CASE iWorkStep OF
	0:		// Powrót do stanu początkowego (ustawienie zmiennych)
		bResetMethod := bQReady := bQBusy := bQError := FALSE;
		IF NOT bLock AND NOT bRelease THEN
			fbTON(IN:= FALSE);
			stInOuts.bAnvilValve := FALSE;
			iWorkStep := 1;
		END_IF
			
	1: 		// Sprawdzenie czy siłowniki są w dobrej pozycji itp.
			IF stInOuts.bLeftActuatorHome AND stInOuts.bRightActuatorHome  THEN
				bQLocked := FALSE;
				iWorkStep := 5;
			END_IF
	
	5:		// Oczekiwanie na nowy rozkaz
			bResetMethod:= bReleaseMethod:= bAuxOperMethod:= bLockMethod := FALSE;
			bQReady := TRUE;
			actCheckForNewOrder();
		
	10:		// Blokowanie kowadła
		IF bEnCheck AND iCtr_SensorWorkVerification > 2 THEN
			nQErrorId := nStFix_NoWeldLock_ErrorCodes.SensorWorkError;
			iWorkStep := 90;
		ELSIF (fbEnclosureSensorFilter.Q OR NOT bEnCheck) AND stInOuts.bLeftActuatorHome AND stInOuts.bRightActuatorHome THEN
			stInOuts.bAnvilValve := TRUE;
			fbTON(IN:= FALSE);
			iWorkStep := 12;	
		ELSIF NOT fbEnclosureSensorFilter.Q AND bEnCheck THEN
			nQErrorId := nStFix_S17EnclosureWelding_ErrorCodes.PartNotDetectedInFixture;
			iWorkStep := 90;
		ELSIF NOT stInOuts.bLeftActuatorHome OR NOT stInOuts.bRightActuatorHome THEN
			nQErrorId := nStFix_S17EnclosureWelding_ErrorCodes.HomePositionMissing;
			iWorkStep := 90;
		END_IF
		
	12: 	// Oczekiwanie na dociśnięcie obudowy
		fbTON(IN:= TRUE,PT:= T#4S);
		IF NOT stInOuts.bLeftActuatorHome AND NOT stInOuts.bRightActuatorHome AND stInOuts.bAnvilBottom THEN	
			bQBusy := FALSE;
			nQErrorId := 0;
			iWorkStep := 5;
		ELSIF fbTON.ET > T#2S AND (stInOuts.bLeftActuatorHome OR stInOuts.bRightActuatorHome) THEN
			nQErrorId := nStFix_S17EnclosureWelding_ErrorCodes.NoMachineReactionOnStartSig;
			iWorkStep := 90;
		ELSIF fbTON.Q THEN
			nQErrorId := nStFix_S17EnclosureWelding_ErrorCodes.TargetPositionTimeout;
			iWorkStep := 90;
		END_IF
		IF iWorkStep <> 12 THEN fbTON(IN:= FALSE); END_IF
		
	20:		// Dodatkowa operacja	
		bPartWelded:= bLastOperStatus;
		IF bEnCheck THEN
			iCtr_SensorWorkVerification := iCtr_SensorWorkVerification + 1;
		END_IF
		bQBusy := FALSE;
		iWorkStep := 5;
		

	30:	// Kowadło zwolnianie
		stInOuts.bAnvilValve:= FALSE;
		fbTON(IN:= FALSE);
		iWorkStep := 32;
		
	32:	// Oczekiwanie na pozycję domową
		fbTON(IN:= TRUE,PT:= T#5S);
		IF stInOuts.bLeftActuatorHome AND stInOuts.bRightActuatorHome AND NOT stInOuts.bAnvilBottom THEN
			bQBusy := FALSE;
			bQLocked := FALSE;		
			iWorkStep := 5;
		ELSIF fbTON.Q THEN
			nQErrorId := nStFix_S17EnclosureWelding_ErrorCodes.BasePositionTimeout;
			iWorkStep := 90;
		END_IF
		IF iWorkStep <> 32 THEN fbTON(IN:= FALSE); END_IF
		
	90:		// Błąd w pracy kowadła
		bQBusy := FALSE;
		bQError := TRUE;
		iWorkStep := 91;
		
	91:
		IF bRelease OR bResetMethod THEN
			iCtr_SensorWorkVerification := 0;
			stInOuts.bAnvilValve := FALSE;
			bQError := FALSE;
			nQErrorId := 0;
			iWorkStep := 0;
		END_IF
		
	ELSE
		mNewEvent(nStFix_S17EnclosureWelding_ErrorCodes.ProgramConfigError);		
END_CASE

END_FUNCTION_BLOCK

// ProdLineMachines/Sonictech/SerialCom/fbSonictechSerialCom
FUNCTION_BLOCK fbSonictechSerialCom IMPLEMENTS I_SonicTech_SerialCom
VAR CONSTANT
	uiMAX_QUEUE_SIZE: UINT := 10;
END_VAR
VAR_IN_OUT
	stData:stSerialComData;
END_VAR
VAR_INPUT
	tTimeout:TIME := T#2S;		// Timeout komunikacji 
	uiResendQty :UINT := 1;			// Liczba ponownych wysłań komend
END_VAR
VAR_OUTPUT
END_VAR
VAR
	fbSerialRead: fbSonictechSerialRcv;
	astCmdsQueue: ARRAY[1..uiMAX_QUEUE_SIZE] OF POINTER TO stSonicTech_SerialCMD;
	bQueueEmpty: BOOL := TRUE;
	bQueueFull: BOOL;
	uiLastCmdIndex: UINT;
	pPtr2ActCmd : POINTER TO stSonicTech_SerialCMD;
	pstDriverData: POINTER TO stSonicTech_SerialStructSoftVer;
	psActProgName: POINTER TO STRING(16);
	pstParametersRange: POINTER TO stSonicTech_SerialStructGenParamsRange;
	pstActualProgramParameters: POINTER TO stSonicTech_SerialStructProgParams;
	pstLastWeldParameters: POINTER TO stSonicTech_SerialStructWeldParams;
	stTestCmdData: stSonicTech_SerialCMD;
	sTestSerialNb: STRING(15);
	stTestDriverData: stSonicTech_SerialStructSoftVer;
	stTestParametersRange: stSonicTech_SerialStructGenParamsRange;
	stTestActualProgramParameters: stSonicTech_SerialStructProgParams;
	stTestLastWeldParameters: stSonicTech_SerialStructWeldParams;
	sTestActProgName: STRING(16);
	byTestActualSonicTechProgNb: BYTE;
	byErrorCode, byTestErrorCode: BYTE;
	// Odbiór danych RS232 
	i: INT;		// Indeks używany w pętlach
	abBufor_Send: ARRAY [1..80] OF BYTE;
	abBufor_String: ARRAY [0..MAX_STRING_LENGTH] OF BYTE;
	bSumaKontrolnaZapytania: BYTE;
	fbSendData:SendData;
	sActProgName2: STRING(16);
	ptPointerToINT:POINTER TO INT;
	ptPointerToUINT:POINTER TO UINT;
	fbTON_RcvTimeout: TON;
	
// Inne	
	nCmdType: nSonicTech_SerialCmdClasses;
	iRozmiarBufora: INT;
	nRecvFrameType: nSonicTech_SerialCmdType;
	bSendCmd: BOOL;				// Bit ustawiany gdy trzeba wysłać rozkaz - kasowany po zakończeniu wysyłania OK bądź NOK
	bWaitingForResponse: BOOL;		// Bit ustawiany po pozytywnym wysłaniu komendy - kasowany po odbiorze danych 
	bReSendCommand: BOOL;		// W razie błędu spróbuj ponownie wysłać komendę
	bCmdExecError: BOOL;	// Błąd w przetwarzaniu komedny
	enComSendErrorMem: Tc2_SerialCom.ComError_t;
	fbClearBuffers:ClearComBuffer;
	bLongExecuteCmd: BOOL;
	fbTONResetComm: TON;
	rCommandReadMeanTime: REAL;
	iComErrors: INT;
	uiReSended: UINT;
	bComReset: BOOL;
	
	bCmdEndedOK: BOOL;
	bAddTestCmd: BOOL;
	nTestCmdType: nSonicTech_SerialCmdClasses;
	fbTON_ComTime: TON;
	bSendTestData: BOOL;
	bPtrsChanged: BOOL;
	bTestCmdFailed: BOOL;
	rLastCmdExecTime: REAL;
	bSendError: BOOL;
	sLastProgName: STRING(255);
	udi_SencCmdCtr: UDINT;
	ui: UINT;
END_VAR

(* ********* Obsługa komunikacji *********
	Nowe zapytanie możliwe gdy typ zapytania=0, jeśli chcemy wykonać zapytanie zmieniamy wartość iTypZapytanie na pożądaną wartość.
	Pętla poniżej zgodnie z typem zapytania przygotowuje zapytanie oraz ustawia flagę bSend.
	Blok wysyłania danych w reakcji na bSend wysyła dane, jeśli wysłanie danych powiodło się, resetuje flagę bSend oraz ustawia bOczekiwanieNaOdpowiedź
	Blok odbierający dane monitoruje zbocze narastające na zmiennej bOczekiwanieNaOdpowiedź, gdy będzie R_TRIG resetuje wewnętrzne dane, ustawia flagę bBusy oraz odbiera dane od zgrzewarki
	Jeśli odbiór był OK wystawia sygnał bDataRecived, jeśli nie wystawia sygnał błędu oraz zeruję flagę bBusy.
*)

ACT_Test_Cmds();
IF nCmdType = nSonicTech_SerialCmdClasses.NoCMD THEN		// Oczekiwanie na nową komendę:
	IF astCmdsQueue[1] <> 0 AND NOT bComReset THEN		// Pobranie nowej komendy z kolejki 
		bLongExecuteCmd := bSendCmd := bWaitingForResponse := FALSE;
		bCmdEndedOK := bCmdExecError := FALSE;
		nCmdType := astCmdsQueue[1]^.nCmdType;
		pPtr2ActCmd := astCmdsQueue[1]; 
		pPtr2ActCmd^.bDone := pPtr2ActCmd^.bError := pPtr2ActCmd^.bSended := FALSE;
	END_IF		
ELSIF bCmdEndedOK OR bCmdExecError THEN			// Sprawdzenie wyniku przetwarzania komendy
	bWaitingForResponse := FALSE;
	fMeanFilter(rInputValue := TIME_TO_REAL(fbTONResetComm.ET), rDelta := 10.0, rMeanValue := rCommandReadMeanTime);
	IF pPtr2ActCmd <> 0 THEN
		pPtr2ActCmd^.bDone := TRUE;
		IF bCmdEndedOK THEN
			pPtr2ActCmd^.nCmdStatus := nSonicTech_SerialCmdStatus.CmdSucceed;
		ELSE
			pPtr2ActCmd^.bError := TRUE;
			pPtr2ActCmd^.nCmdStatus := nSonicTech_SerialCmdStatus.CmdError;	
		END_IF
	END_IF
	pPtr2ActCmd := 0;
	nCmdType := nSonicTech_SerialCmdClasses.NoCMD;
	
	// Sprawdzenie czy są nowe komendy do wykonania
	IF astCmdsQueue[2] <> 0 THEN	// Jest komenda
		MEMMOVE(srcAddr := ADR(astCmdsQueue[2]), destAddr := ADR(astCmdsQueue[1]), n := (uiMAX_QUEUE_SIZE-1)*SIZEOF(astCmdsQueue[2]));
		astCmdsQueue[uiLastCmdIndex]:= 0;
		uiLastCmdIndex := uiLastCmdIndex -1;
		bQueueFull := FALSE;
	ELSE
		astCmdsQueue[1] := 0;
		uiLastCmdIndex := 0;
		bQueueEmpty := TRUE;
	END_IF
END_IF

// Timeout
FOR ui := 2 TO uiLastCmdIndex BY 1 DO
	IF astCmdsQueue[ui] <> 0 THEN
		IF (GVL_Aircom.stAC_DT_Data.tActualTime - astCmdsQueue[ui]^.tTimeStamp) > tTimeout THEN	// Timeout in queue
			astCmdsQueue[ui]^.bDone := astCmdsQueue[ui]^.bError := TRUE;
			astCmdsQueue[ui]^.nCmdStatus := nSonicTech_SerialCmdStatus.CmdError;
			MEMMOVE(srcAddr:= ADR(astCmdsQueue[ui+1]), destAddr := ADR(astCmdsQueue[ui]), n :=(uiLastCmdIndex - ui)*SIZEOF(astCmdsQueue[1]));
			ui := ui -1;	// Ręczna korekta inkrementacji zmiennej w FOR
		END_IF
	END_IF
END_FOR

CASE nCmdType OF
	nSonicTech_SerialCmdClasses.NoCMD:	// Bezczynność
	
	nSonicTech_SerialCmdClasses.ReadSerialNb:	
		IF NOT bSendCmd AND NOT bWaitingForResponse OR bReSendCommand THEN
			abBufor_Send[4]:= 16#00;		// Kod funkcji 0x00 - odczyt numeru seryjnego sterownika
			mFillSendBuffor(Frame := nSonicTech_SerialCmdType.SD1);
			nRecvFrameType := nSonicTech_SerialCmdType.SD2;	
			bSendCmd := TRUE;
		ELSIF fbSerialRead.bDataReceived THEN				// Odbiór danych
			sTestSerialNb := '';
//			fbSerialRead.abBufor_Recv[2] := LIMIT(4,fbSerialRead.abBufor_Recv[2],249);
			IF pPtr2ActCmd <> 0 AND_THEN pPtr2ActCmd^.uiExchangeDataSize >= (fbSerialRead.abBufor_Recv[2]-3) THEN
				MEMCPY(srcAddr := ADR(fbSerialRead.abBufor_Recv[8]),destAddr := pPtr2ActCmd^.pExchangeData, n := (fbSerialRead.abBufor_Recv[2]-3));
				bCmdEndedOK:= TRUE;
			END_IF
			bWaitingForResponse := FALSE;
		END_IF

 	nSonicTech_SerialCmdClasses.ReadMaxParamsValues:	
		IF NOT bSendCmd AND NOT bWaitingForResponse OR bReSendCommand THEN
			abBufor_Send[4]:= 16#01;		// Kod funkcji 0x01 - odczyt zakresu parametrów
			mFillSendBuffor(Frame := nSonicTech_SerialCmdType.SD1);
			nRecvFrameType := nSonicTech_SerialCmdType.SD2;	
			bSendCmd := TRUE;
		ELSIF fbSerialRead.bDataReceived  THEN				// Odbiór danych
			IF pPtr2ActCmd <> 0 AND_THEN pPtr2ActCmd^.uiExchangeDataSize = SIZEOF(stTestParametersRange) THEN
				pstParametersRange := pPtr2ActCmd^.pExchangeData;
				pstParametersRange^.byGeneratorType := fbSerialRead.abBufor_Recv[8];
				ptPointerToUINT := ADR(fbSerialRead.abBufor_Recv[9]);
				pstParametersRange^.uiMinGenFrequency := ROL(ptPointerToUINT^, 8);
				ptPointerToUINT := ADR(fbSerialRead.abBufor_Recv[11]);
				pstParametersRange^.uiMaxGenFrequency := ROL(ptPointerToUINT^, 8);
				ptPointerToUINT := ADR(fbSerialRead.abBufor_Recv[13]);
				pstParametersRange^.uiMaxGenPower := ROL(ptPointerToUINT^, 8);
				ptPointerToUINT := ADR(fbSerialRead.abBufor_Recv[15]);
				pstParametersRange^.uiEncoderLength := ROL(ptPointerToUINT^, 8);
				bCmdEndedOK:= TRUE;
			END_IF
			bWaitingForResponse := FALSE;
		END_IF

	nSonicTech_SerialCmdClasses.ReadSoftVer:	
		IF NOT bSendCmd AND NOT bWaitingForResponse OR bReSendCommand THEN
			abBufor_Send[4]:= 16#03;		// Kod funkcji 0x03 - odczyt wersji oprogramowania
			mFillSendBuffor(Frame := nSonicTech_SerialCmdType.SD1);
			nRecvFrameType := nSonicTech_SerialCmdType.SD3;
			bSendCmd := TRUE;
		ELSIF fbSerialRead.bDataReceived  THEN				// Odbiór danych
			IF pPtr2ActCmd <> 0 AND_THEN pPtr2ActCmd^.uiExchangeDataSize = SIZEOF(stTestDriverData) THEN
				pstDriverData := pPtr2ActCmd^.pExchangeData;
				pstDriverData^.byDriverModel := fbSerialRead.abBufor_Recv[5];
				pstDriverData^.byMajorVersion := fbSerialRead.abBufor_Recv[6];
				pstDriverData^.byMinorVersion := fbSerialRead.abBufor_Recv[7];
				ptPointerToINT := ADR(fbSerialRead.abBufor_Recv[8]);
				pstDriverData^.iBuildNumber := ptPointerToINT^;
				bCmdEndedOK:= TRUE;
			END_IF
		//	sSoftwareVersion := CONCAT(BYTE_TO_STRING(stDaneSterZgrzew.byMajorVersion),CONCAT('.',CONCAT(BYTE_TO_STRING(stDaneSterZgrzew.byMinorVersion),CONCAT('.',INT_TO_STRING(stDaneSterZgrzew.iBuildNumber)))));
			bWaitingForResponse := FALSE;
		END_IF

	nSonicTech_SerialCmdClasses.ReadProgNb:	
		IF NOT bSendCmd AND NOT bWaitingForResponse OR bReSendCommand THEN
			abBufor_Send[4]:= 16#10;		// Kod funkcji 0x10 - odczyt numeru aktualnego programu
			mFillSendBuffor(Frame := nSonicTech_SerialCmdType.SD1);
			nRecvFrameType := nSonicTech_SerialCmdType.SD3;	
			bSendCmd := TRUE;
		ELSIF fbSerialRead.bDataReceived  THEN				// Odbiór danych
			IF pPtr2ActCmd <> 0 AND_THEN pPtr2ActCmd^.uiExchangeDataSize = SIZEOF(byTestActualSonicTechProgNb) THEN
				pPtr2ActCmd^.pExchangeData^ := fbSerialRead.abBufor_Recv[5];
				bCmdEndedOK:= TRUE;
			END_IF
			bWaitingForResponse := FALSE;
		END_IF
			
	nSonicTech_SerialCmdClasses.SetProgNb:
		IF pPtr2ActCmd <> 0 AND_THEN NOT bSendCmd AND NOT bWaitingForResponse OR bReSendCommand THEN
			abBufor_Send[4]:= 16#10;		// Kod funkcji 0x10 - odczyt numeru aktualnego programu
//			MEMCPY(srcAddr := pPtr2ActCmd^.pExchangeData, destAddr := ADR(abBufor_Send[5]) , n := pPtr2ActCmd^.uiExchangeDataSize);
			abBufor_Send[5]:= pPtr2ActCmd^.pExchangeData^;		// Numer aktualnego programu
			MEMSET(destAddr := ADR(abBufor_Send[6]),fillByte:= 0, n:= 7);	// Zerowanie pozostałych bajtów
			mFillSendBuffor(Frame := nSonicTech_SerialCmdType.SD3);
			nRecvFrameType := nSonicTech_SerialCmdType.SC;		
			bSendCmd := TRUE;
		ELSIF fbSerialRead.bDataReceived  THEN				// Odbiór danych
			bCmdEndedOK:= TRUE;
			bWaitingForResponse := FALSE;
		END_IF
			
	nSonicTech_SerialCmdClasses.ReadProgName:
		IF NOT fbSendData.Busy AND NOT bSendCmd AND NOT bWaitingForResponse OR bReSendCommand THEN
			abBufor_Send[4]:= 16#12;		// Kod funkcji 0x12 - odczyt nazwy aktualnego programu
			MEMSET(destAddr := ADR(abBufor_Send[6]),fillByte:= 0, n:= 7);
			abBufor_Send[5]:= pPtr2ActCmd^.pExchangeData^;		// Numer aktualnego programu
			mFillSendBuffor(Frame := nSonicTech_SerialCmdType.SD3);
			nRecvFrameType := nSonicTech_SerialCmdType.SD2;
			bSendCmd := TRUE;
		ELSIF fbSerialRead.bDataReceived  THEN				// Odbiór danych
			MEMCPY(destAddr := ADR(abBufor_String), srcAddr := ADR(fbSerialRead.abBufor_Recv[9]), n:= SIZEOF(abBufor_String));
			sLastProgName := BYTEARR_TO_MAXSTRING(in:= abBufor_String);
			
//			MEMSET(destAddr := ADR(sActProgName2), n := SIZEOF(sActProgName2), fillByte := 0);
//			MEMCPY(destAddr := ADR(sActProgName2), srcAddr := ADR(abBufor_Recv[9]), n:= SIZEOF(sActProgName2)-1);
//			IF pPtr2ActCmd^.uiExchangeDataSize = SIZEOF(sActProgName2) THEN
//				MEMCPY(srcAddr := ADR(sActProgName2), destAddr := pPtr2ActCmd^.pExchangeData, n := pPtr2ActCmd^.uiExchangeDataSize);
//				bCmdEndedOK:= TRUE;
//			END_IF
			bWaitingForResponse := FALSE;
		END_IF

	nSonicTech_SerialCmdClasses.SetProgName:
		IF NOT fbSendData.Busy AND NOT bSendCmd AND NOT bWaitingForResponse OR bReSendCommand THEN
			abBufor_Send[1]:= 16#68;		// Nagłówek zapytania SD2
			abBufor_Send[2]:= 00;		// Ilość danych od DA do końca
			abBufor_Send[3]:= 00;		// Ilość danych od DA do końca
			abBufor_Send[4]:= 16#68;		// Nagłówek zapytania SD3
			abBufor_Send[5]:= pPtr2ActCmd^.bySerialAddr;		// Adres zgrzewarki (domyślnie 51 (0x33)
			abBufor_Send[6]:= 1;			// Adres nadawcy
			abBufor_Send[7]:= 16#12;		// Kod funkcji 0x11 - zapis parametrów aktualnego programu ( 0x13 - Zapis do EEPROM) 
			MEMCPY(srcAddr := pPtr2ActCmd^.pExchangeData, destAddr := ADR(abBufor_Send[8]) , n := pPtr2ActCmd^.uiExchangeDataSize);		// Kolejność jak poniżej 1 +16 bajtów
			//abBufor_Send[8]:= byActualSonicTechProgNb;		// Numer aktualnego programu
			//MEMCPY(srcAddr := ADR(sActProgName2), destAddr := ADR(abBufor_Send[9]), n := 16); 
			bSumaKontrolnaZapytania := 0;				// Obliczanie sumy kontrolnej zapytania
			FOR i:= 5 TO 24 BY 1 DO				// Suma wartości bajtów od DA do FC - dla ramnki SD1
				bSumaKontrolnaZapytania := bSumaKontrolnaZapytania + abBufor_Send[i];
			END_FOR 
			abBufor_Send[25]:= bSumaKontrolnaZapytania;
			abBufor_Send[26]:= 16#16;		// Koniec zapytania - ED
			iRozmiarBufora := 26;				// Rozmiar danych do wysłania
			nRecvFrameType := nSonicTech_SerialCmdType.SC;
			bSendCmd := TRUE;
		ELSIF fbSerialRead.bDataReceived  THEN				// Odbiór danych		
			bCmdEndedOK:= TRUE;	
			bWaitingForResponse := FALSE;
		END_IF
				
	nSonicTech_SerialCmdClasses.ReadProgParams:
		IF NOT fbSendData.Busy AND NOT bSendCmd AND NOT bWaitingForResponse OR bReSendCommand THEN
			abBufor_Send[4]:= 16#11;		// Kod funkcji 0x11 - odczyt parametrów aktualnego programu
			//abBufor_Send[5]:= byActualSonicTechProgNb;		// Numer aktualnego programu
			MEMSET(destAddr := ADR(abBufor_Send[6]),fillByte:= 0, n:= 7);
			mFillSendBuffor(Frame := nSonicTech_SerialCmdType.SD3);
			nRecvFrameType := nSonicTech_SerialCmdType.SD2;
			bLongExecuteCmd := bSendCmd := TRUE;
		ELSIF fbSerialRead.bDataReceived  THEN				// Odbiór danych
			IF pPtr2ActCmd <> 0 AND_THEN pPtr2ActCmd^.uiExchangeDataSize = SIZEOF(stTestActualProgramParameters) THEN
				pstActualProgramParameters:= pPtr2ActCmd^.pExchangeData;
				pstActualProgramParameters^.byWeldType := fbSerialRead.abBufor_Recv[9];
				ptPointerToINT := ADR(fbSerialRead.abBufor_Recv[10]);			
				pstActualProgramParameters^.iMinWeldTime :=ROL(ptPointerToINT^,8);
				ptPointerToINT := ADR(fbSerialRead.abBufor_Recv[12]);			
				pstActualProgramParameters^.iMaxWeldTime := ROL(ptPointerToINT^,8);
				ptPointerToINT := ADR(fbSerialRead.abBufor_Recv[14]);			
				pstActualProgramParameters^.iMinWeldEnergy := ROL(ptPointerToINT^,8);
				ptPointerToINT := ADR(fbSerialRead.abBufor_Recv[16]);			
				pstActualProgramParameters^.iMaxWeldEnergy := ROL(ptPointerToINT^,8);
				ptPointerToINT := ADR(fbSerialRead.abBufor_Recv[18]);			
				pstActualProgramParameters^.iMinGenPower := ROL(ptPointerToINT^,8);
				ptPointerToINT := ADR(fbSerialRead.abBufor_Recv[20]);			
				pstActualProgramParameters^.iMaxGenPower := ROL(ptPointerToINT^,8);			
				ptPointerToINT := ADR(fbSerialRead.abBufor_Recv[22]);			
				pstActualProgramParameters^.iMinDRM := ROL(ptPointerToINT^,8);
				ptPointerToINT := ADR(fbSerialRead.abBufor_Recv[24]);			
				pstActualProgramParameters^.iMaxDRM := ROL(ptPointerToINT^,8);				
				ptPointerToINT := ADR(fbSerialRead.abBufor_Recv[26]);			
				pstActualProgramParameters^.iMinABS := ROL(ptPointerToINT^,8);
				ptPointerToINT := ADR(fbSerialRead.abBufor_Recv[28]);			
				pstActualProgramParameters^.iMaxABS := ROL(ptPointerToINT^,8);			
				ptPointerToINT := ADR(fbSerialRead.abBufor_Recv[30]);			
				pstActualProgramParameters^.iMinTrigerPoint := ROL(ptPointerToINT^,8);
				ptPointerToINT := ADR(fbSerialRead.abBufor_Recv[32]);			
				pstActualProgramParameters^.iMaxTrigerPoint := ROL(ptPointerToINT^,8);			
				ptPointerToINT := ADR(fbSerialRead.abBufor_Recv[34]);			
				pstActualProgramParameters^.uiMinWeldFrequency := INT_TO_UINT( ROL(ptPointerToINT^,8));
				ptPointerToINT := ADR(fbSerialRead.abBufor_Recv[36]);			
				pstActualProgramParameters^.uiMaxWeldFrequency := INT_TO_UINT( ROL(ptPointerToINT^,8));			
				pstActualProgramParameters^.byGenAmplitude := fbSerialRead.abBufor_Recv[38];
				pstActualProgramParameters^.byTrigeringPressure := fbSerialRead.abBufor_Recv[39];
				pstActualProgramParameters^.byIWeldPressure := fbSerialRead.abBufor_Recv[40];
				pstActualProgramParameters^.bIIWeldPressure_EN := fbSerialRead.abBufor_Recv[41]=1;	
				pstActualProgramParameters^.byIIWeldPressure := fbSerialRead.abBufor_Recv[42];
				ptPointerToINT := ADR(fbSerialRead.abBufor_Recv[43]);			
				pstActualProgramParameters^.iSwitchWeldPressPoint := ROL(ptPointerToINT^,8);
				pstActualProgramParameters^.bHoldPressure_EN := fbSerialRead.abBufor_Recv[45] = 1;
				pstActualProgramParameters^.byHoldPressure := fbSerialRead.abBufor_Recv[46];
				ptPointerToINT := ADR(fbSerialRead.abBufor_Recv[47]);	
				pstActualProgramParameters^.iHoldTime := ROL(ptPointerToINT^,8);			
				pstActualProgramParameters^.bAfterBurstImp_EN := fbSerialRead.abBufor_Recv[49]=1;	
				ptPointerToINT := ADR(fbSerialRead.abBufor_Recv[50]);	
				pstActualProgramParameters^.iAfterBurstImpDelayTime := ROL(ptPointerToINT^,8);			
				ptPointerToINT := ADR(fbSerialRead.abBufor_Recv[52]);	
				pstActualProgramParameters^.iAfterBurstImpTime := ROL(ptPointerToINT^,8);		
				pstActualProgramParameters^.bUSTrigerSource := fbSerialRead.abBufor_Recv[54] = 1;
				ptPointerToINT := ADR(fbSerialRead.abBufor_Recv[55]);	
				pstActualProgramParameters^.iTrigerDelayTime := ROL(ptPointerToINT^,8);			
				pstActualProgramParameters^.bSkanAfterProgChange_EN := fbSerialRead.abBufor_Recv[57] = 1;			
				bCmdEndedOK:= TRUE;
			END_IF
			bWaitingForResponse := FALSE;
		END_IF
	
	nSonicTech_SerialCmdClasses.SetProgParams:
		IF NOT bSendCmd AND NOT bWaitingForResponse OR bReSendCommand THEN
			abBufor_Send[2]:= abBufor_Send[3]:= 53;		// Ilość danych od DA do końca
			abBufor_Send[7]:= 16#11;		// Kod funkcji 0x11 - zapis parametrów aktualnego programu ( 0x13 - Zapis do EEPROM) 
			pstActualProgramParameters := pPtr2ActCmd^.pExchangeData;
			abBufor_Send[8]:= pstActualProgramParameters^.byProgNum;
			abBufor_Send[9]:= pstActualProgramParameters^.byWeldType;
			MEMCPY(destAddr := ADR(abBufor_Send[10]), srcAddr := ADR(pstActualProgramParameters^.iMinWeldTime),n := SIZEOF(INT));
			MEMCPY(destAddr := ADR(abBufor_Send[12]), srcAddr := ADR(pstActualProgramParameters^.iMaxWeldTime),n := SIZEOF(INT));
			MEMCPY(destAddr := ADR(abBufor_Send[14]), srcAddr := ADR(pstActualProgramParameters^.iMinWeldEnergy),n := SIZEOF(INT));
			MEMCPY(destAddr := ADR(abBufor_Send[16]), srcAddr := ADR(pstActualProgramParameters^.iMaxWeldEnergy),n := SIZEOF(INT));
			MEMCPY(destAddr := ADR(abBufor_Send[18]), srcAddr := ADR(pstActualProgramParameters^.iMinGenPower),n := SIZEOF(INT));
			MEMCPY(destAddr := ADR(abBufor_Send[20]), srcAddr := ADR(pstActualProgramParameters^.iMaxGenPower),n := SIZEOF(INT));
			MEMCPY(destAddr := ADR(abBufor_Send[22]), srcAddr := ADR(pstActualProgramParameters^.iMinDRM),n := SIZEOF(INT));
			MEMCPY(destAddr := ADR(abBufor_Send[24]), srcAddr := ADR(pstActualProgramParameters^.iMaxDRM),n := SIZEOF(INT));
			MEMCPY(destAddr := ADR(abBufor_Send[26]), srcAddr := ADR(pstActualProgramParameters^.iMinABS),n := SIZEOF(INT));
			MEMCPY(destAddr := ADR(abBufor_Send[28]), srcAddr := ADR(pstActualProgramParameters^.iMaxABS),n := SIZEOF(INT));
			MEMCPY(destAddr := ADR(abBufor_Send[30]), srcAddr := ADR(pstActualProgramParameters^.iMinTrigerPoint),n := SIZEOF(INT));
			MEMCPY(destAddr := ADR(abBufor_Send[32]), srcAddr := ADR(pstActualProgramParameters^.iMaxTrigerPoint),n := SIZEOF(INT));
			MEMCPY(destAddr := ADR(abBufor_Send[34]), srcAddr := ADR(pstActualProgramParameters^.uiMinWeldFrequency),n := SIZEOF(UINT));
			MEMCPY(destAddr := ADR(abBufor_Send[36]), srcAddr := ADR(pstActualProgramParameters^.uiMaxWeldFrequency),n := SIZEOF(UINT));
			abBufor_Send[38]:= pstActualProgramParameters^.byGenAmplitude;
			abBufor_Send[39]:= pstActualProgramParameters^.byTrigeringPressure;
			abBufor_Send[40]:= pstActualProgramParameters^.byIWeldPressure;
			abBufor_Send[41]:= BOOL_TO_BYTE(pstActualProgramParameters^.bIIWeldPressure_EN);
			abBufor_Send[42]:= pstActualProgramParameters^.byIIWeldPressure;
			MEMCPY(destAddr := ADR(abBufor_Send[43]), srcAddr := ADR(pstActualProgramParameters^.iSwitchWeldPressPoint),n := SIZEOF(INT));
			abBufor_Send[45]:= BOOL_TO_BYTE(pstActualProgramParameters^.bHoldPressure_EN);
			abBufor_Send[46]:= pstActualProgramParameters^.byHoldPressure;
			MEMCPY(destAddr := ADR(abBufor_Send[47]), srcAddr := ADR(pstActualProgramParameters^.iHoldTime),n := SIZEOF(INT));
			abBufor_Send[49]:= BOOL_TO_BYTE(pstActualProgramParameters^.bAfterBurstImp_EN);
			MEMCPY(destAddr := ADR(abBufor_Send[50]), srcAddr := ADR(pstActualProgramParameters^.iAfterBurstImpDelayTime),n := SIZEOF(INT));
			MEMCPY(destAddr := ADR(abBufor_Send[52]), srcAddr := ADR(pstActualProgramParameters^.iAfterBurstImpTime),n := SIZEOF(INT));
			abBufor_Send[54]:= BOOL_TO_BYTE(pstActualProgramParameters^.bUSTrigerSource);
			MEMCPY(destAddr := ADR(abBufor_Send[55]), srcAddr := ADR(pstActualProgramParameters^.iTrigerDelayTime),n := SIZEOF(INT));
			abBufor_Send[57]:= BOOL_TO_BYTE(pstActualProgramParameters^.bSkanAfterProgChange_EN);
		
			mFillSendBuffor(Frame := nSonicTech_SerialCmdType.SD2);
			nRecvFrameType := nSonicTech_SerialCmdType.SC;
			bLongExecuteCmd := bSendCmd := TRUE;
		ELSIF fbSerialRead.bDataReceived  THEN				// Odbiór danych	
			bCmdEndedOK:= TRUE;
			bWaitingForResponse := FALSE;
		END_IF

	nSonicTech_SerialCmdClasses.ReadWeldParams:
		// Przygotowanie zapytania
		IF  NOT bSendCmd AND NOT bWaitingForResponse OR bReSendCommand THEN
			abBufor_Send[4]:= 16#20;		// Kod funkcji 0x20 - odczyt parametrów ostatniego zgrzewu
			mFillSendBuffor(Frame := nSonicTech_SerialCmdType.SD1);
			nRecvFrameType := nSonicTech_SerialCmdType.SD2;
			bSendCmd := TRUE;
		ELSIF fbSerialRead.bDataReceived  THEN				// Odbiór danych
			IF pPtr2ActCmd <> 0 AND_THEN pPtr2ActCmd^.uiExchangeDataSize = SIZEOF(stTestLastWeldParameters) THEN
				pstLastWeldParameters:= pPtr2ActCmd^.pExchangeData;
				pstLastWeldParameters^.byWeldStatus := fbSerialRead.abBufor_Recv[8];
				pstLastWeldParameters^.byProgramNumber := fbSerialRead.abBufor_Recv[9];
				pstLastWeldParameters^.byWeldProgType := fbSerialRead.abBufor_Recv[10];
				ptPointerToINT := ADR(fbSerialRead.abBufor_Recv[11]);
				pstLastWeldParameters^.iWeldTime_ms := ROL(ptPointerToINT^,8);
				ptPointerToINT := ADR(fbSerialRead.abBufor_Recv[13]);
				pstLastWeldParameters^.iWeldEnergy_J := ROL(ptPointerToINT^,8);
				ptPointerToINT := ADR(fbSerialRead.abBufor_Recv[15]);
				pstLastWeldParameters^.iGenPower_W := ROL(ptPointerToINT^,8);
				ptPointerToINT := ADR(fbSerialRead.abBufor_Recv[17]);
				pstLastWeldParameters^.iDRM_mm := ROL(ptPointerToINT^,8);
				ptPointerToINT := ADR(fbSerialRead.abBufor_Recv[19]);
				pstLastWeldParameters^.iABS_mm := ROL(ptPointerToINT^,8);
				ptPointerToINT := ADR(fbSerialRead.abBufor_Recv[21]);
				pstLastWeldParameters^.iDAHT_mm := ROL(ptPointerToINT^,8);
				bCmdEndedOK:= TRUE;
			END_IF
			bWaitingForResponse := FALSE;
		END_IF	
		
	nSonicTech_SerialCmdClasses.ReadErrorCode:
		IF NOT bSendCmd AND NOT bWaitingForResponse OR bReSendCommand THEN		// Przygotowanie danych do zapytania
			abBufor_Send[1]:= 16#10;		// Nagłówek zapytania SD1
			abBufor_Send[2]:= pPtr2ActCmd^.bySerialAddr;		// Adres zgrzewarki (domyślnie 51 (0x33))
			abBufor_Send[3]:= 1;			// Adres nadawcy
			abBufor_Send[4]:= 16#21;		// Kod funkcji 0x03 - odczyt wersji oprogramowania
			bSumaKontrolnaZapytania := 0;				// Obliczanie sumy kontrolnej zapytania
			FOR i:= 2 TO 4 BY 1 DO				// Suma wartości bajtów od DA do FC - dla ramnki SD1
				bSumaKontrolnaZapytania := bSumaKontrolnaZapytania + abBufor_Send[i];
			END_FOR 
			abBufor_Send[5]:= bSumaKontrolnaZapytania;
			abBufor_Send[6]:= 16#16;		// Koniec zapytania - ED
			iRozmiarBufora := 6;				// Rozmiar danych do wysłania
			nRecvFrameType := nSonicTech_SerialCmdType.SD3;
			bSendCmd := TRUE;
		ELSIF fbSerialRead.bDataReceived  THEN				// Odbiór danych
			byErrorCode := fbSerialRead.abBufor_Recv[5];
			pPtr2ActCmd^.pExchangeData^:= byErrorCode;
			bCmdEndedOK:= TRUE;
			bWaitingForResponse := FALSE;
		END_IF
	
	ELSE
		nCmdType := nSonicTech_SerialCmdClasses.NoCMD;
END_CASE

//****** Wysłanie zapytania ********************************************************************
IF (bSendCmd OR fbSendData.Busy) THEN
	bSendError := bReSendCommand := FALSE;
	fbSendData(
		pSendData:= ADR (abBufor_Send),
		Length := INT_TO_UDINT(iRozmiarBufora),
		TXbuffer := stData.TxBufferEL);
	IF bSendCmd AND NOT fbSendData.Busy THEN
		bSendCmd := FALSE;
		udi_SencCmdCtr:= udi_SencCmdCtr + 1; 
		IF fbSendData.Error = ComError_t.COMERROR_NOERROR THEN
			fbSerialRead.bRead := TRUE;
			bWaitingForResponse:=TRUE;
			IF pPtr2ActCmd <> 0 THEN
				pPtr2ActCmd^.bSended := TRUE;	
				pPtr2ActCmd^.nCmdStatus := nSonicTech_SerialCmdStatus.Sended;
			END_IF
		ELSE	// Błąd
			bSendError := TRUE;
			enComSendErrorMem := fbSendData.Error;
		END_IF
	END_IF
END_IF 

//****** Odbiór odpowiedzi ********************************************************************
fbSerialRead(RxBufferEL := stData.RxBufferEL,
	tRcvTimeout := SEL(bLongExecuteCmd,T#300MS, T#600MS),
	nFrameType := nRecvFrameType); 
fbSerialRead.bRead R= fbSerialRead.bBusy;		
	
//****** Błąd  ********************************************************************************
IF nCmdType <> nSonicTech_SerialCmdClasses.NoCMD AND (bSendError OR fbSerialRead.bError) THEN		// Błąd wysyłki lub odczytu danych - powtórz wysyłanie
	bSendCmd := FALSE;
	IF uiReSendQty < uiResendQty THEN
		uiReSended := uiReSended +1;
		bReSendCommand := TRUE;
	ELSE
		bCmdExecError := TRUE;
		bComReset := TRUE;
	END_IF
END_IF

// Jeśli nie odebrano danych przed timeoutem reset komunikacji, wystawienie sygnałów do bloczka odczytującego
fbTONResetComm(IN := NOT fbTONResetComm.Q AND nCmdType <> nSonicTech_SerialCmdClasses.NoCMD, PT:= tTimeout); 
IF bComReset OR fbTONResetComm.Q THEN		// Timeout komunikacjie - przerwij odbiór rozkazu
	iComErrors := iComErrors +1;
	bCmdExecError := TRUE;
	bSendCmd := bReSendCommand := FALSE;
	fbClearBuffers(Buffer := stData.RxBufferEL);
	fbClearBuffers(Buffer := stData.TxBufferEL);
	bComReset := FALSE;
END_IF

ACTION ACT_Test_Cmds:
IF bAddTestCmd AND stTestCmdData.nCmdType = nSonicTech_SerialCmdClasses.NoCMD THEN	// Przygotowanie danych i dodanie do kolejki
	stTestCmdData.bSended := stTestCmdData.bError := stTestCmdData.bDone := FALSE;
	stTestCmdData.bySerialAddr := stTestCmdData.bySerialAddr;
	bTestCmdFailed := bPtrsChanged := bSendTestData := FALSE;
	CASE nTestCmdType OF
			nSonicTech_SerialCmdClasses.ReadSerialNb:	
				sTestSerialNb:= '';
				bSendTestData:= TRUE;
			
			nSonicTech_SerialCmdClasses.ReadMaxParamsValues:	// Brak danych wejściowych	
				MEMSET(destAddr := ADR(stTestParametersRange), n := SIZEOF(stTestParametersRange), fillByte := 0);	
				bSendTestData:= TRUE;
			
			nSonicTech_SerialCmdClasses.ReadSoftVer:	// Brak danych wejściowych	
				MEMSET(destAddr := ADR(stTestDriverData), n := SIZEOF(stTestDriverData), fillByte := 0);
				bSendTestData:= TRUE;
			
			nSonicTech_SerialCmdClasses.SetProgNb:	
				stTestCmdData.pExchangeData := ADR(byTestActualSonicTechProgNb);
				stTestCmdData.uiExchangeDataSize := SIZEOF(byTestActualSonicTechProgNb);
				bSendTestData:= TRUE;
				
			nSonicTech_SerialCmdClasses.ReadProgNb:	// Brak danych wejściowych	
				byTestActualSonicTechProgNb := 255;
				bSendTestData:= TRUE;

			nSonicTech_SerialCmdClasses.SetProgParams:	
				stTestCmdData.pExchangeData := ADR(stTestActualProgramParameters);
				stTestCmdData.uiExchangeDataSize := SIZEOF(stTestActualProgramParameters);
				bSendTestData:= TRUE;

			nSonicTech_SerialCmdClasses.ReadProgParams:
				MEMSET(destAddr := ADR(stTestActualProgramParameters), n := SIZEOF(stTestActualProgramParameters), fillByte := 0);
				bSendTestData:= TRUE;

			nSonicTech_SerialCmdClasses.SetProgName:	
				stTestCmdData.pExchangeData := ADR(sTestActProgName);
				stTestCmdData.uiExchangeDataSize := SIZEOF(sTestActProgName);
				bSendTestData:= TRUE;

			nSonicTech_SerialCmdClasses.ReadProgName:
				MEMSET(destAddr := ADR(sTestActProgName), n := SIZEOF(sTestActProgName), fillByte := 0);
				bSendTestData:= TRUE;
			
			nSonicTech_SerialCmdClasses.ReadWeldParams:	
				MEMSET(destAddr := ADR(stTestLastWeldParameters), n := SIZEOF(stTestLastWeldParameters), fillByte := 0);
				bSendTestData:= TRUE;

			nSonicTech_SerialCmdClasses.ReadErrorCode:	
				byTestErrorCode := 0;
				bSendTestData:= TRUE;
		END_CASE
		IF bSendTestData THEN
			stTestCmdData.nCmdType := nTestCmdType;
			IF mAddToQueue(pPtrToData := ADR(stTestCmdData)) THEN			
				bTestCmdFailed := TRUE;
				bAddTestCmd := FALSE;
			END_IF
		ELSE
			bTestCmdFailed := TRUE;
			bAddTestCmd := FALSE;
		END_IF
ELSIF stTestCmdData.nCmdType <> nSonicTech_SerialCmdClasses.NoCMD AND bSendTestData THEN	// Oczekiwanie na odbiór danych
	fbTON_ComTime(IN:= TRUE,PT:= T#3S);
	IF stTestCmdData.bSended AND NOT bPtrsChanged THEN	// Zmiana wskaźników na dane do odebrania
		CASE stTestCmdData.nCmdType OF
			nSonicTech_SerialCmdClasses.ReadSerialNb:	
				stTestCmdData.pExchangeData := ADR(sTestSerialNb);
				stTestCmdData.uiExchangeDataSize := SIZEOF(sTestSerialNb);
			
			nSonicTech_SerialCmdClasses.ReadMaxParamsValues:
				stTestCmdData.pExchangeData := ADR(stTestParametersRange);
				stTestCmdData.uiExchangeDataSize := SIZEOF(stTestParametersRange);
				
			nSonicTech_SerialCmdClasses.ReadSoftVer:
				stTestCmdData.pExchangeData := ADR(stTestDriverData);
				stTestCmdData.uiExchangeDataSize := SIZEOF(stTestDriverData);
	
			nSonicTech_SerialCmdClasses.SetProgNb:
				stTestCmdData.pExchangeData := 0;
				stTestCmdData.uiExchangeDataSize := 0;

			nSonicTech_SerialCmdClasses.ReadProgNb:
				stTestCmdData.pExchangeData := ADR(byTestActualSonicTechProgNb);
				stTestCmdData.uiExchangeDataSize := SIZEOF(byTestActualSonicTechProgNb);

			nSonicTech_SerialCmdClasses.SetProgParams:	
				stTestCmdData.pExchangeData := 0;
				stTestCmdData.uiExchangeDataSize := 0;

			nSonicTech_SerialCmdClasses.ReadProgParams:
				stTestCmdData.pExchangeData := ADR(stTestActualProgramParameters);
				stTestCmdData.uiExchangeDataSize := SIZEOF(stTestActualProgramParameters);
	
			nSonicTech_SerialCmdClasses.SetProgName:	
				stTestCmdData.pExchangeData := 0;
				stTestCmdData.uiExchangeDataSize := 0;

			nSonicTech_SerialCmdClasses.ReadProgName:
				stTestCmdData.pExchangeData := ADR(sTestActProgName);
				stTestCmdData.uiExchangeDataSize := SIZEOF(sTestActProgName);
	
			nSonicTech_SerialCmdClasses.ReadWeldParams:	
				stTestCmdData.pExchangeData := ADR(stTestLastWeldParameters);
				stTestCmdData.uiExchangeDataSize := SIZEOF(stTestLastWeldParameters);
	
			nSonicTech_SerialCmdClasses.ReadErrorCode:	
				stTestCmdData.pExchangeData := ADR(byTestErrorCode);
				stTestCmdData.uiExchangeDataSize := SIZEOF(byTestErrorCode);
		END_CASE
		bPtrsChanged := TRUE;
	ELSIF stTestCmdData.bDone OR fbTON_ComTime.Q THEN
		bSendTestData := bAddTestCmd := FALSE;
		stTestCmdData.nCmdType := nSonicTech_SerialCmdClasses.NoCMD;
		IF stTestCmdData.bDone AND NOT stTestCmdData.bError THEN
			rLastCmdExecTime:= TIME_TO_REAL(fbTON_ComTime.ET);
		ELSE
			bTestCmdFailed:= stTestCmdData.bError;
		END_IF
	END_IF
ELSE
	fbTON_ComTime(IN:= FALSE);
	stTestCmdData.bDone := FALSE;
END_IF
END_ACTION

// Metoda dodaje do kolejki komunikacji nowe polecenie odczytu/zapisu danych - funkcja zwraca natychmiastowo true gdy dodano rozkaz do kolejki
METHOD PUBLIC mAddToQueue : BOOL
VAR_INPUT
	pPtrToData: POINTER TO stSonicTech_SerialCMD;	// Wskaźnik na strukturę danych w bloczku zgrzewarki
END_VAR
IF pPtrToData <> 0 THEN
	IF NOT bQueueFull THEN
		uiLastCmdIndex := LIMIT(1, uiLastCmdIndex + 1, uiMAX_QUEUE_SIZE);
		astCmdsQueue[uiLastCmdIndex] := pPtrToData;
		astCmdsQueue[uiLastCmdIndex]^.bDone := astCmdsQueue[uiLastCmdIndex]^.bError := FALSE;
		astCmdsQueue[uiLastCmdIndex]^.nCmdStatus := nSonicTech_SerialCmdStatus.Queued;
		astCmdsQueue[uiLastCmdIndex]^.tTimeStamp := GVL_Aircom.stAC_DT_Data.tActualTime;
		astCmdsQueue[uiLastCmdIndex]^.bDone := astCmdsQueue[uiLastCmdIndex]^.bError := astCmdsQueue[uiLastCmdIndex]^.bSended := FALSE;
		mAddToQueue := TRUE;
		bQueueFull S= uiLastCmdIndex = uiMAX_QUEUE_SIZE;
	ELSE
		pPtrToData^.bDone := pPtrToData^.bError := TRUE;
		pPtrToData^.nCmdStatus := nSonicTech_SerialCmdStatus.CmdError;
	END_IF
END_IF
END_METHOD

METHOD INTERNAL mFillSendBuffor : BOOL
VAR_INPUT
	Frame: nSonicTech_SerialCmdType;
END_VAR
// Przed wywołaneim metody trzeba uzupełnić zakres danych do zapytania
CASE Frame OF
	nSonicTech_SerialCmdType.SD1:
		abBufor_Send[1]:= 16#10;		// Nagłówek zapytania SD1
		abBufor_Send[2]:= pPtr2ActCmd^.bySerialAddr;		// Adres zgrzewarki (domyślnie 51 (0x33))
		abBufor_Send[3]:= 1;			// Adres nadawcy
//		abBufor_Send[4]:=	- Kod funkcji (uzupełniany przed wywołaniem metody
		bSumaKontrolnaZapytania := 0;				// Obliczanie sumy kontrolnej zapytania
		FOR i:= 2 TO 4 BY 1 DO				// Suma wartości bajtów od DA do FC - dla ramnki SD1
			bSumaKontrolnaZapytania := bSumaKontrolnaZapytania + abBufor_Send[i];
		END_FOR 
		abBufor_Send[5]:= bSumaKontrolnaZapytania;
		abBufor_Send[6]:= 16#16;		// Koniec zapytania - ED
		iRozmiarBufora := 6;			// Rozmiar danych do wysłania		
	
	nSonicTech_SerialCmdType.SD2:
		abBufor_Send[1]:= 16#68;		// Nagłówek zapytania SD2
		abBufor_Send[4]:= 16#68;		// Nagłówek zapytania SD3
		abBufor_Send[5]:= pPtr2ActCmd^.bySerialAddr;		// Adres zgrzewarki (domyślnie 51 (0x33)
		abBufor_Send[6]:= 1;			// Adres nadawcy
		bSumaKontrolnaZapytania := 0;				// Obliczanie sumy kontrolnej zapytania
		
		FOR i:= 5 TO (abBufor_Send[2]+4) BY 1 DO				// Suma wartości bajtów od DA do FC - dla ramnki SD1
			bSumaKontrolnaZapytania := bSumaKontrolnaZapytania + abBufor_Send[i];
		END_FOR 
		abBufor_Send[58]:= bSumaKontrolnaZapytania;
		abBufor_Send[59]:= 16#16;		// Koniec zapytania - ED
		iRozmiarBufora := abBufor_Send[2]+6;				// Rozmiar danych do wysłania
			
	nSonicTech_SerialCmdType.SD3:
		abBufor_Send[1]:= 16#A2;		// Nagłówek zapytania SD3
		abBufor_Send[2]:= pPtr2ActCmd^.bySerialAddr;		// Adres zgrzewarki (domyślnie 51 (0x33)
		abBufor_Send[3]:= 1;			// Adres nadawcy
	
		bSumaKontrolnaZapytania := 0;				// Obliczanie sumy kontrolnej zapytania
		FOR i:= 2 TO 12 BY 1 DO				// Suma wartości bajtów od DA do FC - dla ramnki SD1
			bSumaKontrolnaZapytania := bSumaKontrolnaZapytania + abBufor_Send[i];
		END_FOR 
		abBufor_Send[13]:= bSumaKontrolnaZapytania;
		abBufor_Send[14]:= 16#16;		// Koniec zapytania - ED
		iRozmiarBufora := 14;				// Rozmiar danych do wysłania	
END_CASE
END_METHOD

END_FUNCTION_BLOCK

// ProdLineMachines/Sonictech/SerialCom/I_SonicTech_SerialCom
INTERFACE I_SonicTech_SerialCom

// Metoda dodaje do kolejki komunikacji nowe polecenie odczytu/zapisu danych - funkcja zwraca natychmiastowo true gdy dodano rozkaz do kolejki
METHOD PUBLIC mAddToQueue : BOOL
VAR_INPUT
	pPtrToData: POINTER TO stSonicTech_SerialCMD;	// Wskaźnik na strukturę danych w bloczku zgrzewarki
END_VAR
END_METHOD

END_INTERFACE

// ProdLineMachines/Sonictech/SerialCom/fbSonictechSerialRcv
FUNCTION_BLOCK fbSonictechSerialRcv
VAR CONSTANT
	uiBufferSize: UINT:= 80;		// Rozmiar bufora na dane
END_VAR
VAR_IN_OUT
	RxBufferEL: ComBuffer;
END_VAR
VAR_INPUT
	bRead:BOOL;				// Oczekiwanie na odbiór nowej komendy
	tRcvTimeout:TIME:= T#500MS;			
	nFrameType: nSonicTech_SerialCmdType;	
END_VAR
VAR_OUTPUT
	bBusy: BOOL;
	bDataReceived:BOOL;
	bError: BOOL;
	iErrorCode: INT;
	uiRS_RcvBytesRecived:UINT;			// Ilość odebranych baitów
	abBufor_Recv: ARRAY [1..uiBufferSize] OF BYTE;
END_VAR
VAR
	// Odbiór danych RS232 
	i: INT;		// Indeks używany w pętlach
	fbRS_Receive:ReceiveByte;
	uiRS_RcvDataIndex: UINT;
	uiRS_RcvSD2DataBytes:UINT;
	byRS_RcvCRC_Value: BYTE;
	byDesiredPrefix: BYTE;
	tTON_Timeout: TON;
	uiEndIndex: UINT;
	bRS_RcvCRC_OK: BOOL;
	bReadMem: BOOL;
	bCheckCRC: BOOL;
	bSufixOK: BOOL;
	bPrefixOK: BOOL;
END_VAR

// NIe można zamienić na CASE-y - zbyt wolne przejścia pomiędzy krokami

bDataReceived := FALSE;
IF bRead AND NOT bReadMem THEN
	bError := bCheckCRC := bSufixOK := bRS_RcvCRC_OK :=FALSE;
	bBusy := TRUE;
	iErrorCode := 0;
	uiRS_RcvDataIndex:=1;
	uiRS_RcvBytesRecived:=0;
	MEMSET(destAddr:= ADR(abBufor_Recv), n := SIZEOF(abBufor_Recv), fillByte := 0);
	CASE nFrameType OF
		nSonicTech_SerialCmdType.SD1:	
			byDesiredPrefix := 16#10;
			uiEndIndex := 6;
		nSonicTech_SerialCmdType.SD2:	
			byDesiredPrefix := 16#68;
		nSonicTech_SerialCmdType.SD3:	
			byDesiredPrefix := 16#A2;
			uiEndIndex := 14;
		nSonicTech_SerialCmdType.SC:	
			byDesiredPrefix := 16#E5;	// Znak potwierdzenia
			uiEndIndex := 1;
	END_CASE
	bRead := FALSE;			
END_IF

// Odbiór danych
IF bBusy THEN
	fbRS_Receive(RxBuffer := RxBufferEL);
	IF fbRS_Receive.Error <> ComError_t.COMERROR_NOERROR THEN
		bBusy := FALSE;
		bError := TRUE;
		iErrorCode := fbRS_Receive.Error;				
	END_IF
	// Wczytaj dane z bufora dopóki są w nim dane
	WHILE bBusy AND fbRS_Receive.ByteReceived AND NOT bError DO
		IF uiRS_RcvDataIndex = 1 THEN		// Sprawdzenie znaku początkowego ramki, potwierdzenie typu ramki
			IF byDesiredPrefix <> fbRS_Receive.ReceivedByte THEN
				bError := TRUE;
				iErrorCode := -2;				
			END_IF
			abBufor_Recv[uiRS_RcvDataIndex] := fbRS_Receive.ReceivedByte;
			IF nFrameType = nSonicTech_SerialCmdType.SC THEN
				uiRS_RcvBytesRecived := 1;
				bBusy := FALSE;
				bDataReceived := bSufixOK := TRUE;
			ELSE	
				uiRS_RcvDataIndex := uiRS_RcvDataIndex +1;
			END_IF
		ELSIF uiRS_RcvDataIndex = 2 AND nFrameType = nSonicTech_SerialCmdType.SD2 THEN		// Sprawdzenie liczby danych do odczytu dla SD2
			uiRS_RcvSD2DataBytes :=fbRS_Receive.ReceivedByte;	
			uiEndIndex := uiRS_RcvSD2DataBytes+6;
			abBufor_Recv[uiRS_RcvDataIndex] := fbRS_Receive.ReceivedByte;	
			uiRS_RcvDataIndex := uiRS_RcvDataIndex +1;
		ELSE	// Odczytuj resztę danych
			abBufor_Recv[uiRS_RcvDataIndex] := fbRS_Receive.ReceivedByte;			// Przepisanie odebranego znaku do bufora
			IF uiRS_RcvDataIndex >= uiEndIndex THEN
				bBusy := FALSE;
			ELSE
				uiRS_RcvDataIndex := uiRS_RcvDataIndex +1;
				IF uiRS_RcvDataIndex > uiBufferSize THEN
					bError := TRUE;
					iErrorCode := -3;
				END_IF
			END_IF
			
		END_IF
		bBusy R= bError;
		IF bBusy THEN		// Kontynuacja odczytu
			fbRS_Receive(RXbuffer:= RxBufferEL);
			IF fbRS_Receive.Error <> ComError_t.COMERROR_NOERROR THEN
				bBusy := FALSE;
				bError := TRUE;
				iErrorCode := fbRS_Receive.Error;				
			END_IF		
		ELSIF NOT bError AND NOT bSufixOK THEN	// Normalne wyjście z pętli
			uiRS_RcvBytesRecived := uiRS_RcvDataIndex;
			bSufixOK := bCheckCRC := abBufor_Recv[uiRS_RcvDataIndex] = 16#16;
		END_IF			
	END_WHILE	
END_IF

// Weryfikacja odpowiedzi
IF bCheckCRC THEN		
	byRS_RcvCRC_Value:= 0;
	CASE nFrameType OF			// Sprawdzenie sumy CRC
		nSonicTech_SerialCmdType.SD1:
			FOR i:= 2 TO 4 BY 1 DO			
				byRS_RcvCRC_Value := byRS_RcvCRC_Value + abBufor_Recv[i];
			END_FOR
			bRS_RcvCRC_OK S= (byRS_RcvCRC_Value = abBufor_Recv[5]);
		nSonicTech_SerialCmdType.SD2:
			IF abBufor_Recv[2] = abBufor_Recv[3] THEN
				FOR i:= 5 TO (4 + abBufor_Recv[2]) BY 1 DO
					byRS_RcvCRC_Value := byRS_RcvCRC_Value + abBufor_Recv[i];
				END_FOR 
				bRS_RcvCRC_OK S= (byRS_RcvCRC_Value = abBufor_Recv[(5 + abBufor_Recv[2])]);	
			END_IF
		nSonicTech_SerialCmdType.SD3:
			FOR i:= 2 TO 12 BY 1 DO
				byRS_RcvCRC_Value := byRS_RcvCRC_Value + abBufor_Recv[i];
			END_FOR 
			bRS_RcvCRC_OK S= (byRS_RcvCRC_Value = abBufor_Recv[13]);	
		nSonicTech_SerialCmdType.SC:	bRS_RcvCRC_OK := TRUE;	
	END_CASE
	IF bRS_RcvCRC_OK THEN
		bDataReceived := TRUE;
	ELSE
		bError := TRUE;
	END_IF
	bCheckCRC := FALSE;
END_IF

bReadMem := bRead;

END_FUNCTION_BLOCK

// ProdLineMachines/Sonictech/Welding Machine/fbSonictechUSWM
{attribute 'reflection'} 
FUNCTION_BLOCK PUBLIC fbSonictechUSWM IMPLEMENTS I_StationMachine
VAR_INPUT
	stDigitalInOut		: REFERENCE TO stSonicTech_DigInOuts;		// Wejścia cyfrowe z wtyczki X3_EXT
	I_Fix				: I_Fixture;
	I_SerialCom			: I_SonicTech_SerialCom;
	// Parametry zgrzewarki
	stMachineSettings	: stSonicTech_MachSettings;
END_VAR
VAR_OUTPUT
	bQOperacjaTrwa: BOOL;				// Informacja, że trwa operacja na stanowisku tj. kowadło zakmknięte, zgrzewarka wykonuje zgrzew oraz wyniki pracy są zapisywane do PIM
	bQZgrzewOK: BOOL;
	nError: nSonicTech_ErrorList;
END_VAR
VAR
	I_PimSystem			: I_PIM;
	fbFilter_Error, fbFilter_Ready: fbBinaryFilter;
	bDaneUaktualnione: BOOL;
	sSoftwareVersion: STRING(10);
	stParamAktProgramu: stSonicTech_SerialStructProgParams;
	stParamOstZgrzewu: stSonicTech_SerialStructWeldParams;
	stSerialComData: stSonicTech_SerialCMD;
	bReadMachineParams: BOOL:=TRUE;
	iReadMachineParamsStep: INT:= 0;
	iRMP_Errors: INT;
	byNumerProgramuAkt: BYTE;
	// Komunikacja
	bOdczytOK: BOOL;
	fbTONError: TON;
	rCommandReadMeanTime: REAL;
	uiStat_WeldsQty, uiStat_WeldsOK_Qty, uiStat_WeldsNOK_Qty, uiStat_ErrorsQty: UINT;
	uiStatMem_WeldsQty, uiStatMem_WeldsOK_Qty, uiStatMem_WeldsNOK_Qty, uiStatMem_ErrorsQty: UINT;
	sActProgName: STRING(20);
	fbTON_ResetTimeout: TON;
	fbTON_ParamsRead: TON;
	uiStat_WeldParamsRead: UINT;
	uiStat_ErrorRead: UINT;
	
	
	iWorkStep: INT;
	bLastReadIsWeldParams: BOOL;
	fbTON_TestStepTimeout: TON;
	
	sSqlCmdExtData: STRING(1000);			// Rozkaz do zapisu danych statusowych
	bSqlExtDataSave: BOOL;					// Bit ustawiany po operacji oznacza, że trzeba zapisać dane rozszerzone, resetowany po próbie zapisu
	bSqlExtDataSavedOK: BOOL;				// Bit info o sukcesie dodania danych do kolejki
	astExtData:	ARRAY [1..9] OF stPIM_ExtDataRow;	// Struktura do zapisu danych zgrzewu 
	udiNbOfSavedOkStatuses,	udiNbOfSavedNokStatuses, udiNbOfSavedOkStatusesMEM, udiNbOfSavedNokStatusesMEM: UDINT;	// Liczniki zapusanych statusów PIM
	
	bFixBusy, bFixError: BOOL;
	nFixError: INT;
	bReadWeldData: BOOL;
	bWeldDataActual: BOOL;
	bSendExtDataToDbAfterRead: BOOL;
	bServiceReset: BOOL;
	bCmdAddedToQueue: BOOL;
	byErrorCodeFromWelder: BYTE;
	bFixtureLocked: BOOL;
	bFixtureError: BOOL;
	iFixErrorCode: INT;
	fbTON_ErrorInLogic: TON;
	fbTON_SerialTimeOut: TON;
	bFixConnected: BOOL;
	bFixtureReady: BOOL;
	bTestOutput	: BOOL;
	fbRTrig_TestOutputs: F_TRIG;
END_VAR

(* Przebiegi czasowe zgrzewarki
							Start			  Zgrzew OK						  Zgrzew NOK				Menu			Wyłączenie
Sygnał gotowości 		- ___|¯|_____|¯¯¯¯¯¯¯|_______________|¯¯¯¯¯¯¯¯¯¯¯¯¯¯¯|_______________|¯¯¯¯¯¯¯¯¯|_____|¯¯¯¯¯¯¯¯¯¯|__________
Sygnał generacji US 	- __________________________|¯¯¯|__________________________________________________________________________
Sygnał błędu		 	- _______|¯|_____________________________________________|¯¯¯¯¯¯¯¯¯¯|___________________________|__________
Sygnał zgrzew OK	 	- __________________________________|¯¯¯¯¯¯¯¯¯¯¯¯¯¯¯¯|_____________________________________________________
Sygnał Reset		 	- _______________________________________________________________|¯¯|______________________________________
*)

// Sprawdzenie konfiguracji
//fbRTRIG_UserLogged(CLK:= stPIMInOut.bUzytkownikZalogowany);

fbTON_ErrorInLogic(IN:= NOT fbTON_ErrorInLogic.Q AND iWorkStep < 90 AND (I_PimSystem.prErrorClassExt = nPIM_EventClasses.Error OR I_PimSystem.prErrorClassExt = nPIM_EventClasses.Alarm), PT:= T#1S);
IF fbTON_ErrorInLogic.Q THEN
	mNewEvent(nEvent:=nSonicTech_ErrorList.ProgramConfigError , nEventClass := nPIM_EventClasses.Alarm);
END_IF

IF I_Fix <> 0 THEN		// Wysłanie informacji o stanie maszyny
	bFixConnected:= TRUE;
	I_Fix.prMachState := I_PimSystem.prCurrentMachineState;
 	I_Fix.prUserLogged := I_PimSystem.prUserLogged;
	I_Fix.prTestMode := I_PimSystem.prTestMode;
	I_Fix.prWeldingActive := stDigitalInOut.bWeldingActive;
	I_Fix.prTestOutputsActive := bTestOutput;
	bFixtureReady := I_Fix.prFixReady;
	bFixtureLocked := I_Fix.prFixLocked;
	bFixtureError := I_Fix.prFixError;
	iFixErrorCode := I_Fix.prFixErrorID;
ELSE
	bFixConnected:= FALSE;
END_IF

// Odczyt aktualnych parametrów zgrzewarki
//IF bReadMachineParams THEN
//	ACT_ReadMachineParams();
//END_IF
fbTON_ParamsRead(IN:= bReadMachineParams, PT:= T#2S);
IF fbTON_ParamsRead.Q THEN
	nError:=nSonicTech_ErrorList.NoError;
END_IF

fbRTrig_TestOutputs(CLK:= bTestOutput);
stDigitalInOut.bResetError R= stDigitalInOut.bWorkPermit R= fbRTrig_TestOutputs.Q;				

// Filtrowanie zmiennych wejściowych
fbFilter_Error(IN:= stDigitalInOut.bErrorActive, tON:= T#150MS, tOFF:= T#50MS); 
fbFilter_Ready(IN:= stDigitalInOut.bReadyToWelding, tON:= T#1S, tOFF:= T#2S);  // Do wykrywania wejścia w menu (porównanie sgynału z siłownika i zbocza opadającego na ready)

// Algorytm pracy
CASE iWorkStep OF
	0:	// Inicjalizacja
		I_PimSystem.mSetNewMachineState(nPIM_MachineStates._0_Initialization);
		stSerialComData.bySerialAddr := stMachineSettings.bySerialAdress;
		bQOperacjaTrwa := stDigitalInOut.bWorkPermit := bQZgrzewOK := FALSE;
		IF I_PimSystem.mSetNewMachineState(nPIM_MachineStates._0_Standby_NotReady) THEN
			iWorkStep := 5;
		END_IF
		
	5:	// Oczekiwanie na nowy zgrzew
		I_PimSystem.mSetNewMachineState(nPIM_MachineStates._2_ReadyForNewOperation);
		stDigitalInOut.bWorkPermit R= NOT bTestOutput;
		IF bFixtureLocked OR bFixtureError THEN
			IF iFixErrorCode <> 0 THEN
				mNewEvent(nEvent:= iFixErrorCode , nEventClass := nPIM_EventClasses.Error);
			ELSE
				mNewEvent(nEvent:= nSonicTech_ErrorList.FixtureError , nEventClass := nPIM_EventClasses.Error);
			END_IF
		END_IF
		
		// Wykryty nowy zgrzew - wystawienie sygnału startu na zewnątrz
		IF stDigitalInOut.bStartInput AND NOT stDigitalInOut.bErrorActive THEN	
			IF I_PimSystem.mSetNewMachineState(nPIM_MachineStates._3_NewOperationStarted) THEN
				bSendExtDataToDbAfterRead := bReadWeldData := bQZgrzewOK := FALSE;
				fbTON_TestStepTimeout(IN:= FALSE);
				iWorkStep := 10;
			END_IF
		ELSIF fbFilter_Error.Q THEN		// Aktywny błąd 
			uiStat_ErrorsQty := uiStat_ErrorsQty +1;
			mNewMachEvent();
		ELSIF NOT fbFilter_Ready.Q AND NOT stDigitalInOut.bStartInput THEN		// Wejście w menu
			iWorkStep := 7;			
		END_IF

	7: // Wejście w menu zgrzewarki lub jej wyłączenie
		IF fbFilter_Ready.Q THEN		// Po wyjściu z menu przejdź do kroku gotowości
			iWorkStep := 0;
		ELSIF fbFilter_Error.Q THEN		// Jeśli po wyjściu odrazu błąd odczytaj kod błędu
			uiStat_ErrorsQty := uiStat_ErrorsQty +1;
			mNewMachEvent();
		ELSIF stDigitalInOut.bWeldingActive THEN	// Pomimo braku sygnały z siłownika był zgrzew - nie ustawione wyjście w zgrzewarce
			mNewEvent(nEvent:=nSonicTech_ErrorList.AUX1OutNotSetUp , nEventClass := nPIM_EventClasses.Alarm);
		END_IF

	
	10:	// Potencjalny nowy zgrzew - oczekiwanie na spełnienie warunków zewnętrznych
		IF I_Fix <> 0 THEN		// Jeśli do wejścia kowadła jest podłączony blok obsłuż kowadło, jeśli nie przejdź dalej
			fbTON_TestStepTimeout(IN:= TRUE, PT:= T#3S);
			IF I_Fix.mLock(bBusy=> bFixBusy, bError => bFixError, nErrorCode => nFixError) THEN		// Wywołanie rozkazu, sprawdzenie wyniku
				IF bFixError THEN
					mNewEvent(nEvent:=nFixError, nEventClass := nPIM_EventClasses.Alarm);
				ELSE
					bQOperacjaTrwa := stDigitalInOut.bWorkPermit := TRUE;
					iWorkStep := 15;
				END_IF
			ELSIF NOT bFixBusy AND fbTON_TestStepTimeout.ET > T#500MS THEN		// kowadło nie gotowe do pracy - brak zwrotnego sygnału pracy
 				mNewEvent(nEvent:=nSonicTech_ErrorList.FixtureNoResponse, nEventClass := nPIM_EventClasses.Alarm);
			ELSIF NOT stDigitalInOut.bStartInput THEN	// Sygnał startu zwolniony przed spełnieniem warunków zewnętrznych - chwilowe wciśnięcie dwustartu
				I_PimSystem.mSetNewMachineState(nPIM_MachineStates._2_ReadyForNewOperation);
				I_Fix.mRelease(bReset:= TRUE);
				iWorkStep := 5;
			ELSIF fbFilter_Error.Q THEN						// Błąd niezwiązany ze zgrzewem
				mNewMachEvent();
			END_IF
			IF fbTON_TestStepTimeout.Q THEN			// Warunki zewnętrzne nie spełnione
				mNewEvent(nEvent:=nSonicTech_ErrorList.ExtCondNotMet, nEventClass := nPIM_EventClasses.Alarm);		// Niezidentyfikowany błąd maszyny
			END_IF
			IF iWorkStep <> 10 THEN fbTON_TestStepTimeout(IN:= FALSE);  END_IF
		ELSE
			bQOperacjaTrwa := stDigitalInOut.bWorkPermit := TRUE;
			iWorkStep := 15;
		END_IF	
		
	15:	// Oczekiwanie na sygnał zgrzewania, błąd lub zwolnienie dwustartu: zgrzew- jeśli jest sygnał gen. US lub jeśli błąd wystąpi po czasie większym niż 250ms;
		// błąd -  błąd wyspąpi w czasie mniejszym niż 250ms; menu jeśli przez dłużczy czas żaden z sygnałów nie nastąpi; oczekiwanie na nowy zgrzew jeśli ponownie jest sygnał gotowości
		fbTON_TestStepTimeout(IN:= TRUE, PT:= T#5S);
		IF stDigitalInOut.bWeldingActive OR (fbFilter_Error.Q AND fbTON_TestStepTimeout.ET >= T#250MS) THEN	// Zgrzew lub sygnał złej wysokości ABS, DRM itp. przed zgrzewem
			I_PimSystem.mSetNewMachineState(nPIM_MachineStates._4_OperationInProgress);
			uiStat_WeldsQty:= uiStat_WeldsQty +1;
			iWorkStep := 20;
		ELSIF stDigitalInOut.bReadyToWelding OR NOT stDigitalInOut.bStartInput THEN						// Zgrzewarka ponownie gotowa - dwustart zwolniony
			IF stMachineSettings.bLockWhenOperationsBreaked THEN
				mNewEvent(nEvent:=nSonicTech_ErrorList.StartSignalToShort, nEventClass := nPIM_EventClasses.Alarm);		// Niezidentyfikowany błąd maszyny
			ELSE
				I_PimSystem.mSetNewMachineState(nPIM_MachineStates._2_ReadyForNewOperation);
				bQOperacjaTrwa := stDigitalInOut.bWorkPermit := FALSE;
				iWorkStep := 5;
				IF I_Fix <> 0 THEN
					I_Fix.mRelease(bReset := TRUE);
				END_IF
			END_IF
		END_IF
		IF iWorkStep <> 15 THEN fbTON_TestStepTimeout(IN:= FALSE); END_IF
				
	20:	// Nowy zgrzew trwa - oczekujemy na sygnał zgrzew OK lub sygnał błędu 
		fbTON_TestStepTimeout(IN:= TRUE, PT:= T#20S);
		IF stDigitalInOut.bWeld_OK THEN		// Zgrzew zakończony OK
			bQZgrzewOK := TRUE;
			uiStat_WeldsOK_Qty:= uiStat_WeldsOK_Qty +1;	
			IF I_Fix <> 0 THEN
				I_Fix.mAuxOper(bOperStatus := TRUE);
			END_IF
			iWorkStep := 25;		// Jeśli zgrzew zostanie zakończony i jest komunikacja to przejdź do odczytu parametrów zgrzewu
		ELSIF fbFilter_Error.Q THEN				// Zgrzew zakończony błędem
			uiStat_WeldsNOK_Qty:= uiStat_WeldsNOK_Qty +1;
			IF I_Fix <> 0 THEN
				I_Fix.mAuxOper(bOperStatus := FALSE);
			END_IF
			IF stMachineSettings.bSerialCommunicationEN THEN
				bReadWeldData := TRUE;
				iWorkStep := 35;
			ELSE
				mNewEvent(nEvent:=nSonicTech_ErrorList.UndefinedError, nEventClass := nPIM_EventClasses.Error);	
			END_IF		
		ELSIF fbTON_TestStepTimeout.Q THEN				// Timeout zgrzewu - coś  jest nie tak
			IF NOT stDigitalInOut.bReadyToWelding AND stDigitalInOut.bWeld_OK THEN		// USzkodzony transoptor Ready To Welding
				mNewEvent(nEvent:=nSonicTech_ErrorList.OutputErrorReady, nEventClass := nPIM_EventClasses.Alarm);
			ELSIF stDigitalInOut.bReadyToWelding AND NOT stDigitalInOut.bErrorActive AND NOT stDigitalInOut.bWeld_OK THEN		// USzkodzony transoptor Weld OK
				mNewEvent(nEvent:=nSonicTech_ErrorList.OutputErrorWeldOk, nEventClass := nPIM_EventClasses.Alarm);				
			ELSIF NOT stDigitalInOut.bErrorActive AND NOT stDigitalInOut.bReadyToWelding AND NOT stDigitalInOut.bWeld_OK THEN		// USzkodzony transoptor Error
				mNewEvent(nEvent:=nSonicTech_ErrorList.OutputErrorError, nEventClass := nPIM_EventClasses.Alarm);
			ELSE
				mNewEvent(nEvent:=nSonicTech_ErrorList.ProgramError, nEventClass := nPIM_EventClasses.Alarm);
			END_IF
		END_IF
		IF iWorkStep <> 25 THEN fbTON_TestStepTimeout(IN:= FALSE); END_IF
		
	25:	// Zezwolenie na odblokowanie kowadła po zgrzewie OK
		IF stDigitalInOut.bReadyToWelding THEN
			bSendExtDataToDbAfterRead := bReadWeldData := stMachineSettings.bSerialCommunicationEN;		// Odczytaj parametry zgrzewu
			I_PimSystem.mSetNewMachineState(nPIM_MachineStates._5_OperationEndedOK);
			iWorkStep := 28;
		END_IF
		
	28:	// Oczekiwanie na zgodę na odblokowanie kowadła
		IF I_PimSystem.mSetNewMachineState(nPIM_MachineStates._6_ReturningToBaseState) THEN
			IF I_Fix <> 0 THEN
				fbTON_TestStepTimeout(IN:= FALSE);
				iWorkStep := 30;
			ELSE
				bQOperacjaTrwa := stDigitalInOut.bWorkPermit := FALSE;
				iWorkStep := 0;
			END_IF
		END_IF
				
	30:	// Przetwarzanie zgrzewu zakończone - przygotuj do nowego zgrzewu
		fbTON_TestStepTimeout(IN:= TRUE, PT:= T#4S);
		IF I_Fix.mRelease(bReset := FALSE, bBusy=> bFixBusy, bError => bFixError, nErrorCode => nFixError) THEN		// Wywołanie rozkazu, sprawdzenie wyniku
			IF bFixError THEN
				mNewEvent(nEvent:=nFixError, nEventClass := nPIM_EventClasses.Alarm);
			ELSE
				bQOperacjaTrwa := stDigitalInOut.bWorkPermit := FALSE;
				iWorkStep := 0;
			END_IF
		ELSIF (NOT bFixBusy AND fbTON_TestStepTimeout.ET > T#1S) OR fbTON_TestStepTimeout.Q THEN		// kowadło nie gotowe do pracy - brak zwrotnego sygnału pracy
			mNewEvent(nEvent:=nSonicTech_ErrorList.FixtureNoResponse, nEventClass := nPIM_EventClasses.Alarm);
		END_IF			
		IF iWorkStep <> 30 THEN fbTON_TestStepTimeout(IN:= FALSE); END_IF
		
	35:	// Oczekiwanie na odbiór danych błędnego zgrzewu
		fbTON_SerialTimeOut(IN:=TRUE,PT:= T#2S);
		IF NOT bReadWeldData THEN
			IF bWeldDataActual AND byErrorCodeFromWelder > 0 THEN
				mNewEvent(nEvent:=byErrorCodeFromWelder, nEventClass := nPIM_EventClasses.Error);	
			ELSE
				mNewMachEvent();	//nEvent:=nSonicTech_ErrorList.UndefinedError, nEventClass := nPIM_EventClasses.Error);							
			END_IF
		ELSIF fbTON_SerialTimeOut.Q THEN
			IF GVL_Aircom.bSonicTechSerialComDebug THEN
				mNewEvent(nEvent:=nSonicTech_ErrorList.UndefinedError, nEventClass := nPIM_EventClasses.Error);
			ELSE
				mNewEvent(nEvent:=nSonicTech_ErrorList.Communication_error, nEventClass := nPIM_EventClasses.Error);	
			END_IF
		END_IF 
		IF iWorkStep <> 35 THEN fbTON_SerialTimeOut(IN:= FALSE); END_IF
		
	85: // Odczyt kodu błędu - brak zgrzewu
		IF I_SerialCom <> 0 THEN
			IF NOT bCmdAddedToQueue THEN
				byErrorCodeFromWelder := 0;
				uiStat_ErrorRead := uiStat_ErrorRead +1;
				stSerialComData.nCmdType := nSonicTech_SerialCmdClasses.ReadErrorCode;
				stSerialComData.pExchangeData := ADR(byErrorCodeFromWelder);
				stSerialComData.uiExchangeDataSize := SIZEOF(byErrorCodeFromWelder);
				bCmdAddedToQueue S= I_SerialCom.mAddToQueue(pPtrToData := ADR(stSerialComData));
			ELSE
				IF stSerialComData.bDone AND NOT stSerialComData.bError THEN
					IF byErrorCodeFromWelder <> 0 AND byErrorCodeFromWelder <> 127 AND byErrorCodeFromWelder <> 128 THEN
						mNewEvent(nEvent:=byErrorCodeFromWelder, nEventClass := nPIM_EventClasses.Error);
					ELSIF byErrorCodeFromWelder = 0 AND fbFilter_Error.Q THEN	// Jeśli zwrócony kod błędu wynosi 0 a wyjście błędu aktywne być może uszkodzony transoptor
						mNewEvent(nEvent:=nSonicTech_ErrorList.OutputErrorError, nEventClass := nPIM_EventClasses.Error);
					ELSE	// Jeśli błędy 127 lub 128 wróć do oczekiwania na nowy zgrzew
						IF I_Fix <> 0 THEN
							I_Fix.mRelease(bReset := TRUE);	
						END_IF
						iWorkStep := 0;
					END_IF
				ELSIF stSerialComData.bError OR fbTON_SerialTimeOut.Q THEN
					IF GVL_Aircom.bSonicTechSerialComDebug THEN
						mNewEvent(nEvent:=nSonicTech_ErrorList.UndefinedError, nEventClass := nPIM_EventClasses.Error);
					ELSE
						mNewEvent(nEvent:=nSonicTech_ErrorList.Communication_error, nEventClass := nPIM_EventClasses.Error);	
					END_IF
				END_IF
				fbTON_SerialTimeOut(IN:=TRUE,PT:= T#2S);
			END_IF
			IF iWorkStep <> 85 THEN	 bCmdAddedToQueue := FALSE; fbTON_SerialTimeOut(IN:=FALSE); END_IF		
		ELSE
			mNewEvent(nEvent:=nSonicTech_ErrorList.ProgramConfigError, nEventClass := nPIM_EventClasses.Error);
		END_IF
		
	90:	// WYsterowanie w przypadku błędu
		fbTON_ResetTimeout(IN := FALSE);
		bQZgrzewOK := stDigitalInOut.bWorkPermit := FALSE;
		stDigitalInOut.bResetError := bQOperacjaTrwa := FALSE;
		uiStat_ErrorsQty := uiStat_ErrorsQty +1;
		I_PimSystem.mSetNewMachineState(nPIM_MachineStates._8_WaitForReset);
		iWorkStep := 91;

	91:	// Oczekiwanie na reset
		IF I_PimSystem.mSetNewMachineState(nPIM_MachineStates._9_ResetInProgress) OR bServiceReset THEN
			bServiceReset := FALSE;
			fbTON_ResetTimeout(IN:= FALSE);
			iWorkStep := 95;	
		END_IF
			
	95: // Potwierdzenie błędu itp
		IF NOT fbTON_ResetTimeout.IN AND I_Fix <> 0 THEN
			I_Fix.mRelease(bReset := TRUE);
		END_IF
		stDigitalInOut.bResetError := fbTON_ResetTimeout.ET < T#100MS AND stDigitalInOut.bErrorActive;
		IF stDigitalInOut.bReadyToWelding AND NOT stDigitalInOut.bErrorActive THEN
			nError := nSonicTech_ErrorList.NoError;
			stDigitalInOut.bResetError := FALSE;
			I_PimSystem.mSetNewMachineState(nPIM_MachineStates._0_Standby_NotReady);
			iWorkStep := 0;
		END_IF
		IF fbTON_ResetTimeout.Q THEN
			stDigitalInOut.bResetError := FALSE;
			mNewEvent(nEvent:=nSonicTech_ErrorList.ResetTimeout, nEventClass := nPIM_EventClasses.Alarm);
		END_IF	
		fbTON_ResetTimeout(IN := TRUE, PT:= T#3S);
		
	ELSE
		mNewEvent(nEvent:=nSonicTech_ErrorList.ProgramConfigError, nEventClass := nPIM_EventClasses.Alarm);
END_CASE


IF bReadWeldData THEN			// Odczyt danych zgrzewu
	bWeldDataActual:= FALSE;
	IF I_SerialCom <> 0 THEN
		byErrorCodeFromWelder := 0;
		IF NOT bCmdAddedToQueue THEN
			fbTON_SerialTimeOut(IN:=FALSE);
			uiStat_WeldParamsRead := uiStat_WeldParamsRead +1;
			stSerialComData.nCmdType := nSonicTech_SerialCmdClasses.ReadWeldParams;
			stSerialComData.pExchangeData := ADR(stParamOstZgrzewu);
			stSerialComData.uiExchangeDataSize := SIZEOF(stParamOstZgrzewu);
			IF I_SerialCom.mAddToQueue(pPtrToData := ADR(stSerialComData)) THEN
				bCmdAddedToQueue := TRUE;
			ELSE
				bReadWeldData := FALSE;
			END_IF
		ELSE
			IF stSerialComData.bDone THEN
				bCmdAddedToQueue := bReadWeldData := FALSE;
				IF NOT stSerialComData.bError THEN
					bWeldDataActual := TRUE;
					bSqlExtDataSave := bSendExtDataToDbAfterRead;	
				ELSE
					IF NOT GVL_Aircom.bSonicTechSerialComDebug THEN
						mNewEvent(nEvent:=nSonicTech_ErrorList.Communication_error, nEventClass := nPIM_EventClasses.Alarm);		
					END_IF
				END_IF
			END_IF
		END_IF
		fbTON_SerialTimeOut(IN:=TRUE,PT:= T#2S);
		IF fbTON_SerialTimeOut.Q THEN
			bCmdAddedToQueue := bReadWeldData := FALSE;
			fbTON_SerialTimeOut(IN:=FALSE);
		END_IF
	ELSE
		bReadWeldData := FALSE;
	END_IF
END_IF

IF bSqlExtDataSave THEN			// Zapis danych PIM
	astExtData[1].sName := 'WeldStatus';
	astExtData[1].sValue := BYTE_TO_STRING(stParamOstZgrzewu.byWeldStatus);
	astExtData[2].sName := 'ProgNb';
	astExtData[2].sValue := BYTE_TO_STRING(stParamOstZgrzewu.byProgramNumber);
	astExtData[3].sName := 'WeldMode';
	astExtData[3].sValue := BYTE_TO_STRING(stParamOstZgrzewu.byWeldProgType);
	astExtData[4].sName := 'WeldTime[ms]';
	astExtData[4].sValue := INT_TO_STRING(stParamOstZgrzewu.iWeldTime_ms);
	astExtData[5].sName := 'WeldEnergy[J]';
	astExtData[5].sValue := INT_TO_STRING(stParamOstZgrzewu.iWeldEnergy_J);
	astExtData[6].sName := 'WeldMaxPower[W]';
	astExtData[6].sValue:= INT_TO_STRING(stParamOstZgrzewu.iGenPower_W);
	astExtData[7].sName := 'DRM[mm]';
	astExtData[7].sValue := REAL_TO_STRING(INT_TO_REAL(stParamOstZgrzewu.iDRM_mm)/100.0);
	astExtData[8].sName := 'ABS[mm]';
	astExtData[8].sValue := REAL_TO_STRING(INT_TO_REAL(stParamOstZgrzewu.iABS_mm)/100.0);
	astExtData[9].sName := 'DAHT[mm]';
	astExtData[9].sValue := REAL_TO_STRING(INT_TO_REAL(stParamOstZgrzewu.iDAHT_mm)/100.0);
	bSqlExtDataSavedOK := I_PimSystem.m_SqlInsertExtendedData(pParameters := ADR(astExtData), uiArraySize := SIZEOF(astExtData));
	bSqlExtDataSave := FALSE;	
END_IF


// Statystyka
IF GVL_Aircom.stAC_DT_Data.bNew_Shift THEN
	udiNbOfSavedOkStatusesMEM:= udiNbOfSavedOkStatuses;
	udiNbOfSavedNokStatusesMEM := udiNbOfSavedNokStatuses;
	udiNbOfSavedOkStatuses := udiNbOfSavedNokStatuses := 0;
	uiStatMem_WeldsQty:= uiStat_WeldsQty;
	uiStatMem_WeldsOK_Qty:= uiStat_WeldsOK_Qty;
	uiStatMem_WeldsNOK_Qty:= uiStat_WeldsNOK_Qty;
	uiStatMem_ErrorsQty:= uiStat_ErrorsQty;
	uiStat_WeldParamsRead := uiStat_WeldParamsRead; 
	uiStat_ErrorRead := uiStat_ErrorRead;
	uiStat_WeldsQty:= 0;
	uiStat_WeldsOK_Qty:= 0;
	uiStat_WeldsNOK_Qty:= 0;
	uiStat_ErrorsQty:= 0;
	uiStat_WeldParamsRead := 0; 
	uiStat_ErrorRead := 0;
END_IF

// Kasowanie fixtury w przypadku gdy odłącozno ją od bloku FB
I_Fix := 0;
I_SerialCom := 0;

METHOD FB_init : BOOL
VAR_INPUT
	bInitRetains : BOOL; // if TRUE, the retain variables are initialized (warm start / cold start)
	bInCopyCode : BOOL;  // if TRUE, the instance afterwards gets moved into the copy code (online change)
	I_Pim		: I_PIM;
END_VAR
I_PimSystem := I_Pim;
I_Fix := 0;	// Clear fixture interface - protection against blind interface
END_METHOD

(* Metoda TRUE kiedy dane wyjściowe są ok, jeśli nie FALSE (jeśli not bBusy i FALSE to błąd odczytu) *)
METHOD mGetParamsData : BOOL
VAR_INPUT
	bTestParams:	BOOL;	// Jeśli TRUE metoda okresla czy ma dostęp do parametrów, jeśli tak zwraca TRUE, jeśli nie FALSE
END_VAR
VAR_OUTPUT
	bBusy	: BOOL;										//	Maszyna odświeża dane
	pMachineParametersStruct	: POINTER TO BYTE;		// 	Wskaźnik do parametrów pracy maszyny
	uiMachineParametersSize	: UINT;						// 	Rozmiar struktury parametrów pracy maszyny [bajty]
	wActualCRC16SumInMachine	: WORD;					//	Aktualna suma CRC16 obliczona z parametrów
END_VAR
IF bTestParams THEN
	mGetParamsData := stMachineSettings.bSerialCommunicationEN;
ELSE
	pMachineParametersStruct := ADR(stParamAktProgramu);
	uiMachineParametersSize := SIZEOF(stParamAktProgramu);
	wActualCRC16SumInMachine := F_DATA_TO_CRC16_CCITT(pData := pMachineParametersStruct, cbData := uiMachineParametersSize, crc := 16#0000);
	bBusy := FALSE;
	mGetParamsData := TRUE;	
END_IF
END_METHOD

METHOD INTERNAL mNewEvent : BOOL
VAR_INPUT
	nEventClass:nPIM_EventClasses;
	nEvent: nSonicTech_ErrorList;
END_VAR
bQZgrzewOK := FALSE;
stDigitalInOut.bWorkPermit := FALSE;
IF nEventClass = nPIM_EventClasses.AlarmAutoConfirm OR nEventClass = nPIM_EventClasses.Message THEN		// Alarm nieblokadowy
	I_PimSystem.mSetNewMachineState(nPIM_MachineStates._0_Initialization);
	iWorkStep := 90;
ELSE
	I_PimSystem.mSetNewMachineState(nPIM_MachineStates._7_ErrorOccurr);

	I_PimSystem.mNewEvent(iEventId := nEvent, nEventType := nEventClass, tMessageTime := T#0S);
	iWorkStep := 90;
END_IF
nError := nEvent;
END_METHOD

METHOD INTERNAL mNewMachEvent : BOOL		// Zboczne narastające na wejściu błędu - zareaguj
VAR_INPUT
END_VAR
bQZgrzewOK := FALSE;
stDigitalInOut.bWorkPermit := FALSE;
IF stMachineSettings.bSerialCommunicationEN THEN	
	iWorkStep := 85; 		// Odczytaj kod błędu
	uiStat_ErrorsQty := uiStat_ErrorsQty +1;
ELSE
	mNewEvent(nEvent:=nSonicTech_ErrorList.UndefinedError, nEventClass := nPIM_EventClasses.Error);		// Niezidentyfikowany błąd maszyny
END_IF
END_METHOD

END_FUNCTION_BLOCK

// SQL/fbSQL_Core
FUNCTION_BLOCK FINAL fbSQL_Core IMPLEMENTS I_SQL_Core
VAR CONSTANT
	iNbOfDbBlockInstances:INT:= 8;		// Liczba instancji które obsługują rozkazy
	iQueueSize:INT:=40;					// Rozmiar kolejki na nowe zgłoszenia
END_VAR
VAR_INPUT
	bEnable: BOOL;
	iMaxActiveNodesNb: INT :=iNbOfDbBlockInstances;
	iResendNbIfError:INT:= 3;
	bKeepConnOpen	: BOOL;				// Jeśli true nie rozłącza z bazą danych bezpośrednio po wykonaniu komendy
	bDisableMySQL	: BOOL;				// Whe true extended oprataion data save is disabled
	tCommTimeout	: TIME:= T#3S;
END_VAR
VAR_OUTPUT
	bConnectionMSSQL_OK:BOOL;
	bEmpty:BOOL:= TRUE;	// Kolejka pusta
	bFull:BOOL;		// Zmienna informująca o pełnej kolejce - nie oznacza, że komenda nie zostanie dodana - zostanie jeśli ma większy priorytet niż ostatnia w kolejce
	iQueueLastCmdIndex: INT;	// Liczba komend w kolejce	
	bMasterError:BOOL:= FALSE;	// Wystąpił błąd który uniemożliwia prawidłową pracę komunikacji z DB
END_VAR
VAR
	bInit:BOOL := TRUE;
	afbCoreNodes:ARRAY [1..iNbOfDbBlockInstances] OF fbSQL_CoreNode;
	stTestData:stSQL_ClientNode; 
	astQueue:ARRAY [1..iQueueSize] OF POINTER TO stSQL_ClientNode;	// Kolejka komend wg priorytetu (największy priorytet pierwszy - indeks 0)
	fbSQLDatabase	: FB_SQLDatabaseEvt	(sNetID := '', tTimeout := T#5S);	// Sprawdzanie połączenia do bazy danych
//	fbMySQLDatabase	: FB_SQLDatabaseEvt	(sNetID := '', tTimeout := T#5S);	
	i: INT;
	// Alarmowanie dla danego stanowiska, uiAlarmLoggingLevel mówi jakiego rodzaju alarmy logować, alarmy są przechowywane w fbAlarmTab.
	uiAlarmLoggingLevel:UINT:= 62;
	fbAlarmTab: fbAlarmSlaveTable;
	// Statistics
	udiSQL_Queries_Poped, udiSQL_Queries_OK, udiSQL_Queries_ERR: UDINT;
	rMeanOkCmdTime, rMeanErrCmdTime: REAL;
	sLastErrorDesc: STRING;
	iActiveNodesNb: INT:= 0;
	bSaveUnQueuedCmds: BOOL;
	iConnectionCheckStep:INT;
	fbTON_TestStepTime:TON;
	iCheckConnectionTrials: INT;
	astHMI_NodesTable: ARRAY [1..iNbOfDbBlockInstances] OF stSQL_HMI_CoreNodesData;
	astHMI_QueueTable:ARRAY [1..iQueueSize] OF stSQL_HMI_QueueData;		
	sAlarmMsg: STRING;
	fbStringFormat:FB_FormatString;
	iConvString1,iConvString2: T_MaxString;
	arTimeStats:ARRAY [1..14] OF REAL;	// Rozmiar odpowiadający liczbie komend
	adiCmdsCtr:ARRAY [1..14] OF DINT;	// Licznik wywołań poszczególnych komend
	iCmdType: INT;
	iConectionTestNodeNb: INT;		// Identyfikator węzła który testuje komunikację z DB
	aiMissedCmds:ARRAY [1..14] OF INT;	// Rozmiar odpowiadający liczbie komend - liczba nie zapisanych komend (zakończone przetwarzanie bez rezultatu OK)
	uiEmptyPtr: UINT;
	bCtrReset: BOOL;
	fbTON_ConnCheckMySQL:TON;	// Sprawdzanie czy połączenie jest ok
	bConnectionMySQL_OK:BOOL;
	iConnMySQLRefreshStep: INT;
	fbTON_RefreshMySQL_StepTime: TON;
	iRefreshConnMySQLTrials: INT;
	fbFilter_Warning, fbFilter_Alarm: fbBinaryFilter;
	fbTOF_CommMonitor: TOF;
	bDatabaseConOpen: BOOL;
	fbLogger:fbTextDataLogger;
	bSaveLogs: BOOL;
END_VAR

(*	Opis działania
Jądro komunikacji z PIM zawiera x węzłów (x - stała "iNbOfDbBlockInstances"), każdy z węzłów przetwarza jeden rozkaz. Węzły pracują niezależnie.
Komenda/dane które mają być wysłane do bazy zapisywane są w kolejce "astQueue", podczas zapisu nowa komenda jest wstawiana na odpowiednie miejsce w kolejce zgodnie ze swoim priorytem.
Obsługiwane są dwa rodzaje komend:
- Z danymi zwrotnymi- czyli te które zwracają prewną wartość z bazy danych (np. ID stanowiska) - Wykonanie tych danych blokuje stanowisko do momentu otrzymania odpowiedzi lub błędu zapytania 
- Bez danych zwrotnych - czyli te które są wysyłane do bazy (np. kod alarmu, liczniki zużycia itp) - Podczas dodawania komend do kolejki jest dynamicznie tworzona ich kopia co pozwala nie blokować stanowiska, po wykonaniu komendy pamięć jest zwalniana

*)

//ToDo
// - Timeout przebywania rozkazu w kolejce zależny od priorytetu
// - Jeśli master error nie dodawaj do kolejki

IF bInit THEN
	MEMSET(destAddr := ADR(astQueue), n := SIZEOF(astQueue), fillByte:= 0);		// Czyszczenie kolejki
	bEmpty := TRUE;
	iConectionTestNodeNb := 1;			
	bFull := bInit := FALSE;
	fbLogger.sNetId := '';
	fbLogger.sDirectoryToSave := CONCAT(STR1:= GVL_Aircom.sLogsPath, STR2:='SQL\');
	fbLogger.sFileNameWithFormat := 'CoreLog.txt';		
END_IF

fbLogger(sNetId := '', sPreambule := GVL_Aircom.stAC_DT_Data.sLogTimeString);
IF bSaveLogs THEN
	bSaveLogs := FALSE;
	fbLogger.mSaveBuffor();
END_IF

// Zanim rozpocznie się komunikacja z DB sprawdzenie czy jest z nią połączenie (switch ethernetowy żyje) 
actConnectionCheck();
iResendNbIfError := LIMIT(0,iResendNbIfError, iNbOfDbBlockInstances);
// Obsługa węzłów do komunikacji z PIM - węzły pracują niezależnie
FOR i:= 1 TO iNbOfDbBlockInstances DO
	// Jeśli węzeł bezczynny a kolejka nie pusta pobierz z kolejki komendę
	IF NOT bEmpty AND afbCoreNodes[i].bReadyForNewCmd AND NOT afbCoreNodes[i].bNewQuery AND bEnable AND (bConnectionMSSQL_OK OR bConnectionMySQL_OK) AND NOT bMasterError AND iActiveNodesNb < iMaxActiveNodesNb THEN	
		afbCoreNodes[i].pCmdData := mPopCmdFromQueue();
		IF afbCoreNodes[i].pCmdData <> 0 THEN
			afbCoreNodes[i].pCmdData^.byExecutingNodeNb := INT_TO_BYTE(i);
			//afbCoreNodes[i].pCmdData^.nCmdState := nSQL_CmdExecState.Poped;
			afbCoreNodes[i].bNewQuery := TRUE;
			iActiveNodesNb := iActiveNodesNb + 1;
			udiSQL_Queries_Poped:= udiSQL_Queries_Poped +1;	
		ELSE
			uiEmptyPtr:= uiEmptyPtr + 1; 
		END_IF
	END_IF
	
	afbCoreNodes[i](iResendNbIfError:= iResendNbIfError, bKeepConnOpen:= bKeepConnOpen, tDisconnectTime:= T#10S, tTimeout:= tCommTimeout);
 	afbCoreNodes[i].bCtrReset S= bCtrReset;
	
	IF afbCoreNodes[i].bDone THEN
		IF afbCoreNodes[i].bError THEN
			// Może dodać funkcję logowania błędnych zapytań
			udiSQL_Queries_ERR:= udiSQL_Queries_ERR +1;	
			IF afbCoreNodes[i].udiLastEventId <> 0 THEN
				m_ErrorAnalysis(udiErrNbr:= afbCoreNodes[i].udiLastEventId);	
			END_IF
			sAlarmMsg := CONCAT(STR1 := 'SQL error station: ', STR2 :=afbCoreNodes[i].pCmdData^.sStation );
			sAlarmMsg := CONCAT(STR1 := sAlarmMsg, STR2:= ', cmd: ');
			sAlarmMsg := CONCAT(STR1 := sAlarmMsg, STR2 := TO_STRING(afbCoreNodes[i].pCmdData^.nCmdType));
			sAlarmMsg := CONCAT(STR1 := sAlarmMsg, STR2 := ', ExecTime[s]: ');
			sAlarmMsg := CONCAT(STR1 := sAlarmMsg, STR2 := REAL_TO_STRING(afbCoreNodes[i].rLastExecTimeS) );
			fbAlarmTab.mPushRow(nAlarmClass:= enAlarmClasses.Error, sMachineId := 'PIM Core', sEventDesc := sAlarmMsg , dwErrorId := UDINT_TO_DWORD(afbCoreNodes[i].udiLastEventId));	
			fbLogger.mAddLine(sTextToSave := sAlarmMsg );
			
			iCmdType:= afbCoreNodes[i].pCmdData^.nCmdType;
			IF iCmdType >=1 AND iCmdType <= 14 THEN
				aiMissedCmds[iCmdType] := aiMissedCmds[iCmdType] + 1;
				IF iCmdType = 7 THEN
					fMeanFilter(rInputValue:= afbCoreNodes[i].rLastExecTimeS, rDelta := 10.0,	rMeanValue:= rMeanErrCmdTime);
				END_IF
			END_IF	
		ELSE
			udiSQL_Queries_OK:= udiSQL_Queries_OK +1;	
			// Zbieranie statystyk czasowych
			iCmdType:= afbCoreNodes[i].pCmdData^.nCmdType;
			IF iCmdType >=1 AND iCmdType <= 14 THEN
				adiCmdsCtr[iCmdType] := adiCmdsCtr[iCmdType] + 1;
				fMeanFilter(rInputValue:= afbCoreNodes[i].rLastExecTimeS, rDelta := 10.0,	rMeanValue:= arTimeStats[iCmdType]);
				IF iCmdType = 7 THEN
					fMeanFilter(rInputValue:= afbCoreNodes[i].rLastExecTimeS, rDelta := 10.0,	rMeanValue:= rMeanOkCmdTime);
				END_IF
			END_IF
			
		END_IF
		
		// Zakończenie przetwarzania rozkazu
		IF NOT afbCoreNodes[i].pCmdData^.bWaitForDataReturn THEN// Jeśli rozkaz wygenerowany dynamicznie zwolnij zaalokowaną pamięć
			__DELETE(afbCoreNodes[i].pCmdData);
		END_IF 		
		afbCoreNodes[i].pCmdData := 0;
		iActiveNodesNb := LIMIT(0,iActiveNodesNb - 1,iNbOfDbBlockInstances);
		afbCoreNodes[i].bNewQuery := FALSE;
	END_IF		
	
		
	// Dane do HMI rdzenie
	IF GVL_Aircom.stAC_DT_Data.bNew_Second_IMP THEN
		astHMI_NodesTable[i].iNumber := i;
		astHMI_NodesTable[i].bBusy := afbCoreNodes[i].bBusy;
		astHMI_NodesTable[i].bHangUp := FALSE;
	END_IF
END_FOR

// Dane do HMI kolejka
IF GVL_Aircom.stAC_DT_Data.bNew_Second_IMP THEN
	FOR i := 1 TO iQueueSize DO
		astHMI_QueueTable[i].iNumber := i;
		IF astQueue[i] <> 0 THEN
			astHMI_QueueTable[i].sStationName := astQueue[i]^.sStation;
			astHMI_QueueTable[i].nCmdType := astQueue[i]^.nCmdType;
			astHMI_QueueTable[i].bWaitForDataReturn := astQueue[i]^.bWaitForDataReturn;
		ELSE
			astHMI_QueueTable[i].sStationName := '';
			astHMI_QueueTable[i].nCmdType := nSQL_CmdTypes.None;
			astHMI_QueueTable[i].bWaitForDataReturn := FALSE;
		END_IF
	END_FOR
END_IF
IF bCtrReset THEN
	bCtrReset := FALSE;	
	udiSQL_Queries_Poped:= udiSQL_Queries_OK:= udiSQL_Queries_ERR := 0;
	iActiveNodesNb := 0;
END_IF

// Alarmowanie
fbTOF_CommMonitor(IN:= FALSE,PT:=T#30S);
fbFilter_Warning(IN:= fbTOF_CommMonitor.Q AND (rMeanOkCmdTime > (TIME_TO_REAL(tCommTimeout)*0.0005)),tON:= T#3S, tOFF:= T#10S);
IF fbFilter_Warning.RTrig THEN
	sAlarmMsg := CONCAT(STR1:= CONCAT(STR1 := 'High PIM SQL cmd exec time (>50% timeout):- ', STR2 :=REAL_TO_STRING(rMeanOkCmdTime)), STR2:= '[s]');
	fbAlarmTab.mPushRow(nAlarmClass:= enAlarmClasses.Warning, sMachineId := 'Cmd Exec', sEventDesc := sAlarmMsg , dwErrorId := 0);	
	fbLogger.mAddLine(sTextToSave := sAlarmMsg );					
END_IF
fbFilter_Alarm(IN:= fbTOF_CommMonitor.Q AND (rMeanOkCmdTime > (TIME_TO_REAL(tCommTimeout)*0.0008)),tON:= T#2S, tOFF:= T#10S);
IF fbFilter_Alarm.RTrig THEN
	sAlarmMsg := CONCAT(STR1:= CONCAT(STR1 := 'Critical PIM SQL cmd exec time (>80% timeout):- ', STR2 :=REAL_TO_STRING(rMeanOkCmdTime)), STR2:= '[s]');
	fbAlarmTab.mPushRow(nAlarmClass:= enAlarmClasses.Error, sMachineId := 'Cmd Exec', sEventDesc := sAlarmMsg , dwErrorId := 0);	
	fbLogger.mAddLine(sTextToSave := sAlarmMsg );					
END_IF

ACTION actConnectionCheck:

bDatabaseConOpen := fbSQLDatabase.bConnected;
CASE iConnectionCheckStep OF
	0:		// Oczekiwanie na rozkaz sprawdzenia połączenia
		IF NOT bConnectionMSSQL_OK AND NOT bMasterError AND iConnMySQLRefreshStep = 0 THEN
			iConnectionCheckStep := 5;
			fbTON_TestStepTime(IN:= FALSE);
			iCheckConnectionTrials := 0;
		END_IF
		
	4:		// Oczekiwanie na powtórzenie zapytania
		fbTON_TestStepTime(IN:= TRUE, PT:= T#10S);
		IF fbTON_TestStepTime.Q THEN
			iCheckConnectionTrials:= iCheckConnectionTrials + 1;
			iConnectionCheckStep := 5;
			fbTON_TestStepTime(IN:= FALSE);
		END_IF
	
	5:		// Przygotowanie danych
		IF NOT fbSQLDatabase.bBusy AND NOT bMasterError THEN
			iConnectionCheckStep := 10;					
			fbTON_TestStepTime(IN:= FALSE);
		END_IF

	10:		// Oczekiwanie na zakończenie komendy
		IF fbSQLDatabase.Connect(hDBID := 1) THEN
			bConnectionMSSQL_OK := NOT fbSQLDatabase.bError;
			iConnectionCheckStep := 15;
			
	(*		IF fbSQLDatabase.bError THEN
				fbTON_TestStepTime(IN:= FALSE);
				iConnectionCheckStep := 4;
			ELSE
				bConnectionMSSQL_OK := TRUE;
				iConnectionCheckStep := 15;
			END_IF	*)
		END_IF
		
	15:		// Rozłączenie
		IF fbSQLDatabase.Disconnect() THEN
			IF fbSQLDatabase.bError THEN
				iConnectionCheckStep := 20;		
			ELSE
				IF bConnectionMSSQL_OK THEN
					iConnectionCheckStep := 0;
				ELSE
					iConnectionCheckStep := 4;
				END_IF
			END_IF
		END_IF

	20:	// Sprawdzenie połączenia
		IF fbSQLDatabase.bConnected THEN
			iConnectionCheckStep := 15;
		ELSE
			IF bConnectionMSSQL_OK THEN
				iConnectionCheckStep := 0;
			ELSE
				iConnectionCheckStep := 4;
			END_IF
		END_IF
END_CASE

// Odświeżenie komunikacji z MySQL
fbTON_ConnCheckMySQL(IN:= iConnMySQLRefreshStep = 0, PT:= T#5M);
CASE iConnMySQLRefreshStep OF
	0:		// Oczekiwanie na rozkaz sprawdzenia połączenia
		IF (iConnectionCheckStep = 0 ) AND (NOT bConnectionMySQL_OK OR fbTON_ConnCheckMySQL.Q) THEN
			iConnMySQLRefreshStep := 5;
			iRefreshConnMySQLTrials := 0;
		END_IF
		
	4:		// Oczekiwanie na powtórzenie zapytania
		fbTON_RefreshMySQL_StepTime(IN:= TRUE, PT:= T#10S);
		IF fbTON_RefreshMySQL_StepTime.Q THEN
			iRefreshConnMySQLTrials:= iRefreshConnMySQLTrials + 1;
			iConnMySQLRefreshStep := 5;
			fbTON_RefreshMySQL_StepTime(IN:= FALSE);
		END_IF
	
	5:		// Przygotowanie danych
		IF NOT fbSQLDatabase.bBusy THEN
			iConnMySQLRefreshStep := 10;					
		END_IF

	10:		// Oczekiwanie na zakończenie komendy
		IF fbSQLDatabase.Connect(hDBID := 2) THEN
			bConnectionMySQL_OK := NOT fbSQLDatabase.bError;
			iConnMySQLRefreshStep := 15;
			fbTON_RefreshMySQL_StepTime(IN:= FALSE);
		END_IF

	15:		// Rozłączenie
		IF fbSQLDatabase.Disconnect() THEN
			IF fbSQLDatabase.bError THEN
				iConnMySQLRefreshStep := 20;		
			ELSE
				IF bConnectionMySQL_OK THEN
					iConnMySQLRefreshStep := 0;
				ELSE
					iConnMySQLRefreshStep := 4;
				END_IF
			END_IF
		
		END_IF
		
	20:
		IF fbSQLDatabase.bConnected THEN
			iConnMySQLRefreshStep := 15;
		ELSE
			IF bConnectionMySQL_OK THEN
				iConnMySQLRefreshStep := 0;
			ELSE
				iConnMySQLRefreshStep := 4;
			END_IF
		END_IF
	
END_CASE
END_ACTION

METHOD IsCoreWork : BOOL
VAR_INPUT
END_VAR
IsCoreWork := bEnable AND bConnectionMSSQL_OK AND NOT bMasterError;
END_METHOD

METHOD PRIVATE m_ErrorAnalysis : BOOL
VAR_INPUT
	udiErrNbr:UDINT;
END_VAR
				
CASE udiErrNbr OF
	0:		// No error
		sLastErrorDesc:= 'Brak bledu';
	1792:	sLastErrorDesc:= 'Blad ogolny';
	1793:	sLastErrorDesc:= 'Serwis nie obslugiwany przez serwer';
	1794:	sLastErrorDesc:= 'Niewlasciwa grupa';
	1795:	sLastErrorDesc:= 'Niewlasciwy offset';
	1796:	sLastErrorDesc:= 'Odczyt lub zapis niedozwolony';
	1797:	sLastErrorDesc:= 'Niewlasciwy rozmiar parametrow';
	1798:	sLastErrorDesc:= 'Niewlasciwe wartosci zmiennych';
	1799:	sLastErrorDesc:= 'Urzadzenie nie gotowe do pracy';
	1800:	sLastErrorDesc:= 'Urzadzenie zajete';
	1828:	// No license Error
		bMasterError := TRUE;
		sLastErrorDesc:= 'Brak aktywnej licencji';
	ELSE
		sLastErrorDesc:= 'Inny blad';
END_CASE
END_METHOD

// Jeśli dodanie do kolejki poprawne zmienna wyjściowa ma wartość TRUE przy wywołaniu, jeśli nie (błąd dodania) FALSE
METHOD PUBLIC mAddCmdToQueue : BOOL	
VAR_INPUT
	pNewCmdData:POINTER TO stSQL_ClientNode;
END_VAR
VAR_OUTPUT
	nErrorID:nSQL_ErrorCodes;
END_VAR
VAR
	iQueueAddSearchIndex: INT;
END_VAR
IF pNewCmdData <= 0 THEN		//Wykonaj kod tylko jeśli prawidłowy wskaźnik wejściowy,
	mAddCmdToQueue := FALSE;
	nErrorID := nSQL_ErrorCodes.AddBadPointer;
	RETURN;
ELSIF bMasterError THEN
	mAddCmdToQueue := FALSE;
	nErrorID := nSQL_ErrorCodes.AddNewFailedMasterErrorAtCore;
	RETURN;
ELSIF bDisableMySQL AND (pNewCmdData^.nCmdType = nSQL_CmdTypes.InsCompressedAirCons OR pNewCmdData^.nCmdType = nSQL_CmdTypes.InsEnergyCons 
		OR pNewCmdData^.nCmdType = nSQL_CmdTypes.InsExtendedData) THEN
	mAddCmdToQueue := FALSE;
	RETURN;
END_IF	

nErrorID := nSQL_ErrorCodes.NoError;

// Jeśli kolejka jest pusta dodaj na początek listy
IF bEmpty THEN			
	MEMSET(destAddr := ADR(astQueue), n := SIZEOF(astQueue[1]), fillByte:= 0);		// Czyszczenie pozycji
	// Jeśli czeka na dane zwrotne przypisz do kolejki instancję z bloku klienta, jeśli nie wygeneruj dynmiczny blok pamięci i przepisz dane
	IF pNewCmdData^.bWaitForDataReturn THEN		
		astQueue[1] := pNewCmdData;
		astQueue[1]^.nCmdState := nSQL_CmdExecState.Queued;
		mAddCmdToQueue := TRUE;
	ELSE
		astQueue[1] := __NEW(stSQL_ClientNode);
		IF astQueue[1] > 0 THEN
		//	MEMCPY(srcAddr:= pNewCmdData, destAddr := astQueue[1], n := SIZEOF(stPIM_ClientNode));
			astQueue[1]^ := pNewCmdData^;
			mAddCmdToQueue := TRUE;		
			astQueue[1]^.nCmdState := nSQL_CmdExecState.Queued;
		ELSE
			mAddCmdToQueue := FALSE;
			nErrorID := nSQL_ErrorCodes.AddNewOperatorFail;
		END_IF
	END_IF
	bEmpty := FALSE;
	bFull := iQueueSize = 1;	// Aktualizuj zmienne
	iQueueLastCmdIndex := 1;	// Zmienna mówiąca w którym indeksie znajduje się ostatnia komenda 

// Jeśli nie pusta dodaj do kolejki na koniec wg priorytetu (first in first out)
ELSE 		
	iQueueAddSearchIndex := LIMIT(1,iQueueLastCmdIndex,iQueueSize);// Przeszukuj kolejkę od końca
	WHILE iQueueAddSearchIndex > 0 AND_THEN astQueue[iQueueAddSearchIndex]^.nCmdType < pNewCmdData^.nCmdType DO	// Zmniejszanie indeksu dopóki nie znajdzie równego lub wyższego priorytetu
		iQueueAddSearchIndex := iQueueAddSearchIndex - 1;
	END_WHILE
	// po wyjściu z pętli zmienna SearchIndex ma wartość ostatniego elementu o !niemniejszym! priorytecie, na indeks+1 trzeba wprowadzić nową komendę
	
	// Przesunmięcie zadań (przygotowanie miejsca dla nowo wstawianej komendy)
	// Jeśli kolejka nie jest w pełni zapełniona przesuń zadania i nie przejmuj się resztą
	IF iQueueLastCmdIndex < iQueueSize THEN		
		MEMMOVE(srcAddr:= ADR(astQueue[iQueueAddSearchIndex+1]),destAddr := ADR(astQueue[iQueueAddSearchIndex+2]), n:=SIZEOF(astQueue[1])*INT_TO_UINT(iQueueLastCmdIndex-iQueueAddSearchIndex));
		iQueueLastCmdIndex := iQueueLastCmdIndex + 1;	// Zwiększenie indeksu ostatniej komendy
		bFull S= iQueueLastCmdIndex = iQueueSize;		// Sprawdzenie czy kolejka jest pełna
		
	// Jeśli kolejka pełna przesuń o jeden rozkaz mniej (ostatni rozkaz w kolejce nadpisany - jeśłi był wygenerowany automatycznie trzeba go usunąć), jeśli ostatni ma równy priorytet pominń dodanie rozkazu	
	ELSE		
		IF astQueue[iQueueLastCmdIndex]>0 THEN 
			// Przesuń tylko gdy ostatnia komenda ma mniejszy priorytet
			IF astQueue[iQueueLastCmdIndex]^.nCmdType < pNewCmdData^.nCmdType THEN 		
// Miejsce na zapisanie usuwanej komendy
//				IF bSaveUnQueuedCmds THEN
				IF NOT astQueue[iQueueLastCmdIndex]^.bWaitForDataReturn THEN	// Jeśli rozkaz dynamiczny usuń
					__DELETE(astQueue[iQueueLastCmdIndex]);
				ELSE															// Jeśli rozkaz z danymi powrotnymi uaktualnij stan
					astQueue[iQueueLastCmdIndex]^.bSQL_Done := TRUE;
					astQueue[iQueueLastCmdIndex]^.bSQL_OK := FALSE;
					astQueue[iQueueLastCmdIndex]^.nCmdState := nSQL_CmdExecState.UnQueued;					
				END_IF
				IF iQueueAddSearchIndex < (iQueueSize-1) THEN	// Jeśli nowy rozkaz jest wstawiany na miejsce miejsze niż ostatnie przesuń rozkazy, inaczej nic nie rób
					MEMMOVE(srcAddr:= ADR(astQueue[iQueueAddSearchIndex+1]),destAddr := ADR(astQueue[iQueueAddSearchIndex+2]), n:=SIZEOF(astQueue[1])*INT_TO_UINT(iQueueLastCmdIndex-iQueueAddSearchIndex-1));
				END_IF				
			END_IF
		END_IF			
		iQueueLastCmdIndex := iQueueSize;	// Zwiększenie indeksu ostatniej komendy
		bFull := TRUE;
	END_IF
	
	// Wstawienie nowej komendy do kolejki
	IF iQueueAddSearchIndex < iQueueSize THEN
		IF pNewCmdData^.bWaitForDataReturn THEN		// Jeśli czeka na dane zwrotne przypisz do kolejki instancję z bloku klienta
			astQueue[iQueueAddSearchIndex+1] := pNewCmdData;
			astQueue[iQueueAddSearchIndex+1]^.nCmdState := nSQL_CmdExecState.Queued;
			astQueue[iQueueAddSearchIndex+1]^.bSQL_Done := astQueue[iQueueAddSearchIndex+1]^.bSQL_OK := FALSE;
			mAddCmdToQueue := TRUE;
		ELSE	// Jeśli nie wygeneruj dynamicznie blok pamięci i przepisz dane
			astQueue[iQueueAddSearchIndex+1] := __NEW(stSQL_ClientNode);
			IF astQueue[iQueueAddSearchIndex+1] > 0 THEN
				//	MEMCPY(srcAddr:= pNewCmdData, destAddr := astQueue[iQueueAddSearchIndex+1], n := SIZEOF(stPIM_ClientNode));
				astQueue[iQueueAddSearchIndex+1]^ :=pNewCmdData^;
				astQueue[iQueueAddSearchIndex+1]^.nCmdState := nSQL_CmdExecState.Queued;
				astQueue[iQueueAddSearchIndex+1]^.bSQL_Done := astQueue[iQueueAddSearchIndex+1]^.bSQL_OK := FALSE;
				mAddCmdToQueue := TRUE;		
			ELSE
				mAddCmdToQueue := FALSE;
				nErrorID := nSQL_ErrorCodes.AddNewOperatorFail;
			END_IF
		END_IF
	ELSE	// Jeśli brak miejsca w kolejce na rozkaz o danym priorytecie zakończ
		mAddCmdToQueue := FALSE;
		nErrorID := nSQL_ErrorCodes.AddNewNoSpaceForAddPriority;
	END_IF
END_IF
END_METHOD

METHOD PRIVATE mPopCmdFromQueue : POINTER TO stSQL_ClientNode
VAR_INPUT
END_VAR
IF bEmpty OR astQueue[1] = 0 THEN	// Jeśli kolejka pusta pomiń pobranie rozkazu
	mPopCmdFromQueue := 0;
	bEmpty := FALSE;
ELSE			// Jeśli nie pusta pobierz rozkaz
	mPopCmdFromQueue := astQueue[1];// Pobranie wskaźnika z początku kolejki 
	IF iQueueLastCmdIndex > 1 THEN	// Jeśli więcej niż jeden rozkaz w kolejce przesuń kolejkę, zmień indeks ostatniej komendy
		iQueueLastCmdIndex := iQueueLastCmdIndex - 1;	// Aktualizacja liczby rozkazów w kolejce
		MEMMOVE(srcAddr:= ADR(astQueue[2]),destAddr := ADR(astQueue[1]), n:=SIZEOF(astQueue[1])*INT_TO_UINT(iQueueLastCmdIndex));	//Przesunięcie kolejki
		bFull := FALSE;
		astQueue[iQueueLastCmdIndex+1] := 0;	// Wyzerowanie wskaźnika		
	ELSE	// Jeśli w kolejce pozostał jeden rozkaz nie trzeba przesuwać kolejki itp
		astQueue[1] := 0;
		iQueueLastCmdIndex := 0;
		bFull := FALSE;	
		bEmpty := TRUE;
	END_IF
END_IF
END_METHOD

END_FUNCTION_BLOCK

// SQL/fbSQL_CoreNode
FUNCTION_BLOCK fbSQL_CoreNode
VAR_INPUT
	bNewQuery			: BOOL;
	pCmdData			: POINTER TO stSQL_ClientNode;		// Wskaźnik na dane przetwarzanego rozkazu
	iResendNbIfError	: INT:= 2;
	bKeepConnOpen		: BOOL:= FALSE;						// Jeśli TRUE nie zamykaj połączenia
	tDisconnectTime		: TIME;								// Czas po którym nastąpi zamknięcie połączenia do DB w przypadku bezczynności
	tTimeout			: TIME;								// Czas timeout-u
	bCtrReset			: BOOL;								// Reset liczników
END_VAR
VAR_OUTPUT
	bDone				: BOOL;								// Impuls w momencie zakończenia przetwarzania
	bBusy				: BOOL:= FALSE;						// Informacja o zajętości węzła - 0 wolny, 1 zajęty
	bError				: BOOL:= FALSE;						// Błąd przetwarzania
	bReadyForNewCmd		: BOOL;								// Blok gotowy na nową komendę
	rLastExecTimeS		: REAL; 
	udiLastEventId		: UDINT;
END_VAR
VAR
	iResendQty			: INT:= 0;							// Licznik ponownych wysłań komunikatu
	bConnectedToDB		: BOOL;								// Info czy węzęł ma aktywne podłączenie do DB
	iConnectedDBId		: INT;								// Numer bazy danych do podłączenia
	iStep, iLastStep	: INT;								// krok przetwarzania zapytania
	iDB_ID				: INT:= 1;							// Identyfikator bazy danych przez którą powinny być przetwarzane komendy
	fbSQLDatabase		: FB_SQLDatabaseEvt	(sNetID := '', tTimeout := T#5S);	// Zarządzanie połączeniem z bazą danych
	fbSQLCommand		: FB_SQLCommandEvt	(sNetID := '', tTimeout := T#5S);	// Wykonanie komendy
	fbSQLStoredProc		: FB_SQLStoredProcedureEvt	(sNetID := '', tTimeout := T#5S);	// Wykonanie procedury SQL
	fbSQLResult			: FB_SQLResultEvt (sNetID := '', tTimeout := T#5S);		// Odczyt pobranych danych
	fbTON_TimeStats		: TON;								// Timer do statystyk czasowych
	udiSQL_Queries_New, udiSQL_Queries_OK, udiSQL_Queries_ERR: UDINT;
	bResend: BOOL;
	astSP_ParamsDef	: ARRAY [0..5] OF ST_SQLSPParameter;
	fbTON_DisconnectTime: TON;
	bOnlyDisconnect: BOOL;
	fbTON_MasterTimeout: TON;
	iMasterTimeoutCtr: INT;
	sLastEventText: STRING;
	sLastEventClass: STRING;
	sLastDisconnectEventText: STRING;
	sLastDisconnectEventClass: STRING;
	iErrCtr: INT;
	fbFTRig_Disconnect: F_TRIG;
	bSQL_SP: BOOL;
END_VAR

fbTON_DisconnectTime(IN:= fbSQLDatabase.bConnected AND NOT bBusy AND NOT bNewQuery, PT:= tDisconnectTime);
IF GVL_Aircom.bInit THEN
	ACT_Init();
ELSIF pCmdData > 0 AND_THEN bBusy THEN
	pCmdData^.bSQL_LifeBit := TRUE;
END_IF

fbTON_MasterTimeout(IN:= bBusy, PT:=2*tTimeout);
IF fbTON_MasterTimeout.Q THEN
	iMasterTimeoutCtr:= iMasterTimeoutCtr +1; 
END_IF
CASE iStep OF
	0:	// Dodano nową komendę, sprawdź czy połączenie otwarte oraz czy zgadza się numer DB
		bDone := FALSE;
		IF bCtrReset THEN
			bCtrReset := FALSE;
			udiSQL_Queries_New:= udiSQL_Queries_OK:= udiSQL_Queries_ERR:= 0;
		END_IF
		IF pCmdData <> 0 AND_THEN (bNewQuery OR bResend) THEN
			// Uzupełnienie danych komendy
			pCmdData^.nCmdState := nSQL_CmdExecState.Processing;
			pCmdData^.bSQL_Done := pCmdData^.bSQL_OK := FALSE;
			pCmdData^.bSQL_Busy := bBusy := TRUE;
			udiLastEventId := pCmdData^.udiLEventId := 0;
			fbSQLCommand.tTimeout := tTimeout;
			fbSQLDatabase.tTimeout := fbSQLResult.tTimeout := tTimeout/3;
			udiSQL_Queries_New := udiSQL_Queries_New + 1;
			bOnlyDisconnect := bError := FALSE;
			IF NOT bResend THEN
				pCmdData^.sEventText := '';
				iResendQty := 0;
			END_IF
			
			// Wybór bazy do której zostaną zapisane dane
			CASE pCmdData^.nCmdType OF	
				nSQL_CmdTypes.InsCompressedAirCons, nSQL_CmdTypes.InsEnergyCons, nSQL_CmdTypes.InsExtendedData:
  				iDB_ID := 2;
			ELSE
				iDB_ID := 1;
			END_CASE
			
			// SPrawdzenie połączenia
			
			IF fbSQLDatabase.bConnected AND iConnectedDBId = iDB_ID THEN	// Połączenie jest ok, przejdź do wysłania komendy
				iStep := 10;
			ELSIF NOT fbSQLDatabase.bConnected THEN		// podłącz do odpowiedniej bazy danych	
				iStep := 6;
			ELSE	// podłączono do złej bazy danych, rozłącz i podłącz ponownie
				iStep := 4;
			END_IF
			
			bNewQuery := bResend := FALSE;
			fbTON_TimeStats(IN:= TRUE, PT:= T#10S);
		ELSIF fbTON_DisconnectTime.Q THEN
			bOnlyDisconnect := TRUE;
			iStep := 4;
		ELSE
			bReadyForNewCmd := TRUE;
		END_IF;
		bReadyForNewCmd R= iStep > 0;
			
	4:	// Rozłacz połączenie z DB
		iLastStep := iStep;
		IF fbSQLDatabase.Disconnect() THEN
			IF fbSQLDatabase.bError THEN	// Błąd
				mSaveError(I_TcMsg := fbSQLDatabase.ipTcResult);
				sLastDisconnectEventText := sLastEventText;
				sLastDisconnectEventClass := sLastEventClass;
				iStep := 90;		
			ELSE
				iStep := SEL(bOnlyDisconnect,6,0);
			END_IF
		ELSIF NOT fbSQLDatabase.bBusy THEN
			IF pCmdData <> 0 AND_THEN pCmdData^.udiLEventId = 0 THEN
				pCmdData^.udiLEventId := INT_TO_UDINT(iStep);
				pCmdData^.sEventText := 'Fb not busy';				
			END_IF
			iStep := 90;
		END_IF
	
	6:	// Podłącz do odpowiedniej DB
		iLastStep := iStep;
		IF fbSQLDatabase.Connect(hDBID := INT_TO_UDINT(iDB_ID)) THEN
			IF fbSQLDatabase.bError THEN	// Błąd
				mSaveError(I_TcMsg := fbSQLDatabase.ipTcResult);
				iStep := 90;		
			ELSE
				iConnectedDBId := iDB_ID;

				iStep := 10;
			END_IF
		ELSIF NOT fbSQLDatabase.bBusy THEN
			IF pCmdData <> 0 AND_THEN pCmdData^.udiLEventId = 0 THEN
				pCmdData^.udiLEventId := INT_TO_UDINT(iStep);
				pCmdData^.sEventText := 'Fb not busy';				
			END_IF
			iStep := 90;
		END_IF	
		
	10:	// Przygotowanie zapytania - komenda SQL
		iLastStep := iStep;
		bNewQuery := FALSE;
		IF pCmdData^.nCmdType <> nSQL_CmdTypes.SelInsStatusOfOperation AND_THEN 
						fbSQLDatabase.CreateCmd(pSQLCommand := ADR(fbSQLCommand)) THEN
			IF NOT fbSQLDatabase.bError THEN	// Połączenie zlinkowane
				IF pCmdData^.bWaitForDataReturn THEN
					iStep := 20;	// Zapis danych + oczekiwanie na dane zwrotne	
				ELSE
					iStep := 15;	// Zapis danych, bez danych powrtonych
				END_IF												
			ELSE
				mSaveError(I_TcMsg := fbSQLDatabase.ipTcResult);	
				iStep := 90;
			END_IF
		
		ELSIF pCmdData^.nCmdType = nSQL_CmdTypes.SelInsStatusOfOperation AND_THEN 
						fbSQLDatabase.CreateSP(sProcedureName:= '[dbo].[InsertPartStatus]', pParameterInfo := ADR(astSP_ParamsDef) , cbParameterInfo :=SIZEOF(astSP_ParamsDef), pSQLProcedure := ADR(fbSQLStoredProc)) THEN
			IF NOT fbSQLDatabase.bError THEN	// Połączenie zlinkowane
				IF pCmdData^.bWaitForDataReturn THEN
					iStep := 21;	// Zapis danych + oczekiwanie na dane zwrotne	
				ELSE
					iStep := 16;	// Zapis danych, bez danych powrtonych
				END_IF												
			ELSE
				mSaveError(I_TcMsg := fbSQLDatabase.ipTcResult);	
				iStep := 90;
			END_IF
			
		ELSIF NOT fbSQLDatabase.bBusy THEN
			IF pCmdData <> 0 AND_THEN pCmdData^.udiLEventId = 0 THEN
				pCmdData^.udiLEventId := INT_TO_UDINT(iStep);
				pCmdData^.sEventText := 'Fb not busy';				
			END_IF
			iStep := 90;
		END_IF
					
	15:	// Wysłanie komendy typu INSERT - bez danych zwrotnych 
		iLastStep := iStep;
		IF 	fbSQLCommand.Execute(pSQLCmd := ADR(pCmdData^.sCmdExpression),cbSQLCmd := SIZEOF(pCmdData^.sCmdExpression)) THEN
			IF fbSQLCommand.bError THEN
				mSaveError(I_TcMsg := fbSQLCommand.ipTcResult);
				iStep := 90;		
			ELSE
				iStep := 30;
			END_IF
		ELSIF NOT fbSQLCommand.bBusy THEN
			IF pCmdData <> 0 AND_THEN pCmdData^.udiLEventId = 0 THEN
				pCmdData^.udiLEventId := INT_TO_UDINT(iStep);
				pCmdData^.sEventText := 'Fb not busy';				
			END_IF
			iStep := 90;
		END_IF
	
	16:		// Wywołanie procedury bez danych zwrotnych
		IF fbSQLStoredProc.Execute(pParameterStrc := ADR(pCmdData^.stStatusSaveParams),cbParameterStrc := SIZEOF(pCmdData^.stStatusSaveParams)) THEN
			IF fbSQLStoredProc.bError THEN
				mSaveError(I_TcMsg := fbSQLStoredProc.ipTcResult);
				iStep := 90;		
			ELSE
				iStep := 30;
			END_IF
		ELSIF NOT fbSQLStoredProc.bBusy THEN
			IF pCmdData <> 0 AND_THEN pCmdData^.udiLEventId = 0 THEN
				pCmdData^.udiLEventId := INT_TO_UDINT(iStep);
				pCmdData^.sEventText := 'Fb not busy';				
			END_IF
			iStep := 90;
		END_IF
		
	20:	// Wysłanie komendy typu SELECT - pobranie info z DB
		iLastStep := iStep;
		IF fbSQLCommand.ExecuteDataReturn( 
					pSQLCmd:= ADR(pCmdData^.sCmdExpression), 
					cbSQLCmd:= SIZEOF(pCmdData^.sCmdExpression), 
					pSQLDBResult:= ADR(fbSQLResult)) THEN
			IF fbSQLCommand.bError THEN
				mSaveError(I_TcMsg := fbSQLCommand.ipTcResult);
				iStep := 90;		
			ELSE
				iStep := 25;
			END_IF
		ELSIF NOT fbSQLCommand.bBusy THEN
			IF pCmdData <> 0 AND_THEN pCmdData^.udiLEventId = 0 THEN
				pCmdData^.udiLEventId := INT_TO_UDINT(iStep);
				pCmdData^.sEventText := 'Fb not busy';				
			END_IF
			iStep := 90;
		END_IF

	21:	// Wykonanie procedury zwracającej dane wyjściowe - pobranie info z DB
		iLastStep := iStep;
		IF fbSQLStoredProc.ExecuteDataReturn( 
					pParameterStrc:= ADR(pCmdData^.stStatusSaveParams), 
					cbParameterStrc:= SIZEOF(pCmdData^.stStatusSaveParams), 
					pSQLDBResult:= ADR(fbSQLResult)) THEN
			IF fbSQLStoredProc.bError THEN
				mSaveError(I_TcMsg := fbSQLStoredProc.ipTcResult);
				iStep := 90;		
			ELSE
				iStep := 25;
			END_IF
		ELSIF NOT fbSQLStoredProc.bBusy THEN
			IF pCmdData <> 0 AND_THEN pCmdData^.udiLEventId = 0 THEN
				pCmdData^.udiLEventId := INT_TO_UDINT(iStep);
				pCmdData^.sEventText := 'Fb not busy';				
			END_IF
			iStep := 90;
		END_IF
	
	25:	// Pobranie wyniku
		iLastStep := iStep;
		IF fbSQLResult.Read(nStartIndex := 0,
					nRecordCount := 1,
					pData:= pCmdData^.pReturnedData, 
					cbData:= pCmdData^.uiReturnedDataSize, 
					bDataRelease := TRUE,
					bWithVerifying := FALSE) THEN
			IF fbSQLResult.bError THEN
				mSaveError(I_TcMsg := fbSQLResult.ipTcResult);
				iStep := 90;
			ELSE
				fbSQLStoredProc.Release();
				iStep := 30;
			END_IF	
		ELSIF NOT fbSQLResult.bBusy THEN
			IF pCmdData <> 0 AND_THEN pCmdData^.udiLEventId = 0 THEN
				pCmdData^.udiLEventId := INT_TO_UDINT(iStep);
				pCmdData^.sEventText := 'Fb not busy';				
			END_IF
			iStep := 90;
		END_IF		
	
	30:	// Zwolnienie procedury
		IF fbSQLStoredProc.Release() THEN
			iStep := 31;
		END_IF	
				
	31: // Sprawdzenie czy zamknąć połączenie
		iLastStep := iStep;
		IF bKeepConnOpen THEN
			iStep := 32;
		ELSE
			IF fbSQLDatabase.Disconnect() THEN
				IF fbSQLDatabase.bError THEN	// Błąd
					mSaveError(I_TcMsg := fbSQLDatabase.ipTcResult);
					sLastDisconnectEventText := sLastEventText;
					sLastDisconnectEventClass := sLastEventClass;
					iStep := 90;
				ELSE		
					iStep := 32;
				END_IF
			ELSIF NOT fbSQLDatabase.bBusy THEN
				IF pCmdData <> 0 AND_THEN pCmdData^.udiLEventId = 0 THEN
					pCmdData^.udiLEventId := INT_TO_UDINT(iStep);
					pCmdData^.sEventText := 'Fb not busy';				
				END_IF
				iStep := 90;
			END_IF
		END_IF
		
	32:	// Zakończenie przetwarzania rozkazu OK	
		udiSQL_Queries_OK:= udiSQL_Queries_OK +1;	
		pCmdData^.bSQL_Busy := bBusy := bError := FALSE;
		bDone := pCmdData^.bSQL_OK := pCmdData^.bSQL_Done := TRUE;		
		pCmdData^.nCmdState := nSQL_CmdExecState.Succeed;
		fbTON_TimeStats();
		rLastExecTimeS := TIME_TO_REAL(fbTON_TimeStats.ET)/1000;
		fbTON_TimeStats(IN:= FALSE);
		pCmdData^.rCmdExecTimeMS := rLastExecTimeS;
		IF NOT bNewQuery THEN
			iStep := 0;
		ELSE
			iStep := 33;
		END_IF
		
	33:	// Oczekiwanie na reset sygnału wejściowego
		IF NOT bNewQuery THEN
			iStep := 0;
		END_IF
			
	90:	
		udiSQL_Queries_ERR := udiSQL_Queries_ERR +1;	
		IF pCmdData <> 0 THEN
			fbTON_TimeStats();
			rLastExecTimeS := TIME_TO_REAL(fbTON_TimeStats.ET)/1000;
			pCmdData^.rCmdExecTimeMS := rLastExecTimeS;	
		END_IF
		fbTON_TimeStats(IN:= FALSE);
		bError := TRUE;
		IF pCmdData <> 0 AND_THEN iResendQty < iResendNbIfError AND NOT bOnlyDisconnect THEN
			iResendQty := iResendQty +1;
			iStep := 0;
			bResend := TRUE;
			pCmdData^.nCmdState := nSQL_CmdExecState.ReSend;
		ELSE
			IF NOT bKeepConnOpen AND fbSQLDatabase.bConnected THEN
				iStep := 91;
			ELSE 
				iStep := 92;
			END_IF
		END_IF
	
	91: // Zakończenie przetwarzania po błędzie
		IF fbSQLDatabase.Disconnect() THEN
			IF fbSQLDatabase.bError THEN	// Błąd
				mSaveError(I_TcMsg := fbSQLDatabase.ipTcResult);
				sLastDisconnectEventText := sLastEventText;
				sLastDisconnectEventClass := sLastEventClass;
				iStep := 90;		
			ELSE
				iStep := 92;
			END_IF
		ELSIF NOT fbSQLDatabase.bBusy THEN
			IF pCmdData <> 0 AND_THEN pCmdData^.udiLEventId = 0 THEN
				pCmdData^.udiLEventId := INT_TO_UDINT(iStep);
				pCmdData^.sEventText := 'Fb not busy';				
			END_IF
			iStep := 90;
		END_IF

	92:	// Powrót do stanu początkowego
		IF pCmdData <> 0 THEN
			pCmdData^.bSQL_Busy := FALSE;
			pCmdData^.bSQL_Done := TRUE;	
			pCmdData^.nCmdState := nSQL_CmdExecState.Error;
		END_IF
		bBusy := FALSE;	
		bDone := NOT bOnlyDisconnect AND pCmdData <> 0;
		IF NOT bNewQuery THEN
			iStep := 0;
		ELSE
			iStep := 32;
		END_IF		
END_CASE

fbFTRig_Disconnect(CLK:= fbSQLDatabase.bConnected);
IF fbFTRig_Disconnect.Q THEN
	iConnectedDBId := -1;
END_IF

ACTION ACT_Init:
// 0- Id stacji
astSP_ParamsDef[0].sParameterName := '@idLineStation';
astSP_ParamsDef[0].eParameterType := E_SPParameterType.Input;
astSP_ParamsDef[0].eParameterDataType := E_ColumnType.Integer;
astSP_ParamsDef[0].nParameterSize := 4;

// 1- status
astSP_ParamsDef[1].sParameterName := '@status';
astSP_ParamsDef[1].eParameterType := E_SPParameterType.Input;
astSP_ParamsDef[1].eParameterDataType := E_ColumnType.BIT_;
astSP_ParamsDef[1].nParameterSize := 1;

// 2- machineNumber
astSP_ParamsDef[2].sParameterName := '@machineNumber';
astSP_ParamsDef[2].eParameterType := E_SPParameterType.Input;
astSP_ParamsDef[2].eParameterDataType := E_ColumnType.SmallInt;
astSP_ParamsDef[2].nParameterSize := 2;

// 3- isHidden
astSP_ParamsDef[3].sParameterName := '@isHidden';
astSP_ParamsDef[3].eParameterType := E_SPParameterType.Input;
astSP_ParamsDef[3].eParameterDataType := E_ColumnType.BIT_;
astSP_ParamsDef[3].nParameterSize := 1;

// 4- isTest
astSP_ParamsDef[4].sParameterName := '@isTest';
astSP_ParamsDef[4].eParameterType := E_SPParameterType.Input;
astSP_ParamsDef[4].eParameterDataType := E_ColumnType.BIT_;
astSP_ParamsDef[4].nParameterSize := 1;

// 5- Quantity
astSP_ParamsDef[5].sParameterName := '@quantity';
astSP_ParamsDef[5].eParameterType := E_SPParameterType.Input;
astSP_ParamsDef[5].eParameterDataType := E_ColumnType.Float;
astSP_ParamsDef[5].nParameterSize := 8;
END_ACTION

METHOD mSaveError
VAR_INPUT
	I_TcMsg: I_TcMessage;
END_VAR
(*udiLastEventId := I_TcMsg.nEventId;
I_TcMsg.RequestEventText(nLangId := 1033, sResult := sLastEventText, nResultSize := SIZEOF(sLastEventText));
I_TcMsg.RequestEventClassName(nLangId := 1033, sResult := sLastEventClass, nResultSize := SIZEOF(sLastEventClass));	*)
IF pCmdData <> 0 THEN
	pCmdData^.udiLEventId:= 0;//udiLastEventId;
	pCmdData^.sEventText := 'Unknown error';//sLastEventText;
END_IF
END_METHOD

END_FUNCTION_BLOCK

